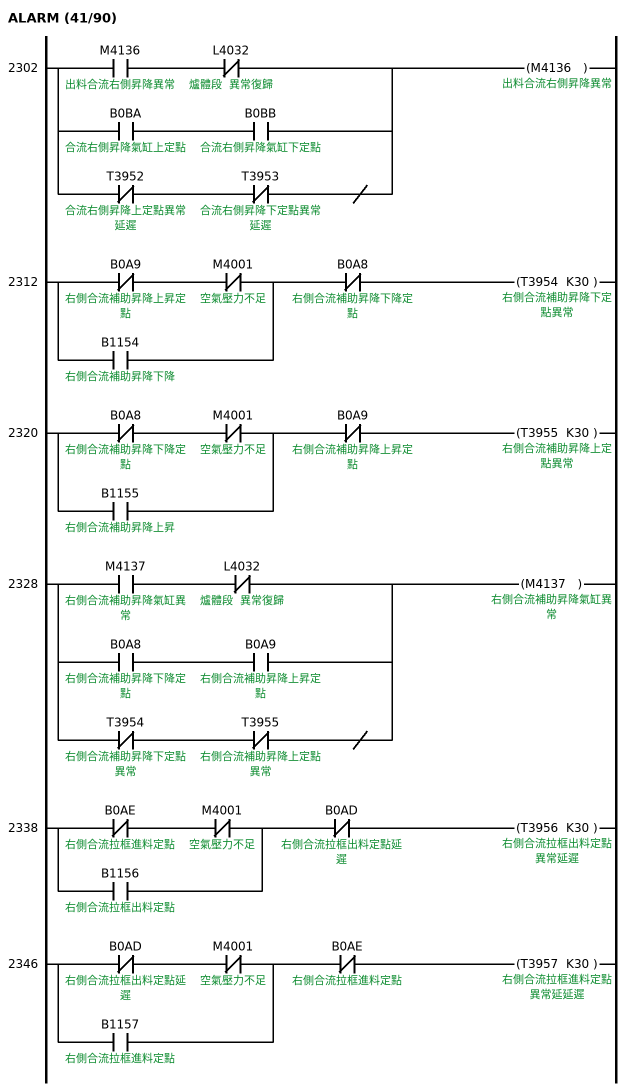
2302  LD      M4136  ; 出料合流右側昇降異常
      ANI     L4032  ; 爐體段  異常復歸
      LD      B0BA  ; 合流右側昇降氣缸上定點
      AND     B0BB  ; 合流右側昇降氣缸下定點
      ORB
      LDI     T3952  ; 合流右側昇降上定點異常延遲
      ANI     T3953  ; 合流右側昇降下定點異常延遲
      INV
      ORB
      OUT     M4136  ; 出料合流右側昇降異常
2312  LDI     B0A9  ; 右側合流補助昇降上昇定點
      ANI     M4001  ; 空氣壓力不足
      OR      B1154  ; 右側合流補助昇降下降
      ANI     B0A8  ; 右側合流補助昇降下降定點
      OUT     T3954 K30  ; 右側合流補助昇降下定點異常
2320  LDI     B0A8  ; 右側合流補助昇降下降定點
      ANI     M4001  ; 空氣壓力不足
      OR      B1155  ; 右側合流補助昇降上昇
      ANI     B0A9  ; 右側合流補助昇降上昇定點
      OUT     T3955 K30  ; 右側合流補助昇降上定點異常
2328  LD      M4137  ; 右側合流補助昇降氣缸異常
      ANI     L4032  ; 爐體段  異常復歸
      LD      B0A8  ; 右側合流補助昇降下降定點
      AND     B0A9  ; 右側合流補助昇降上昇定點
      ORB
      LDI     T3954  ; 右側合流補助昇降下定點異常
      ANI     T3955  ; 右側合流補助昇降上定點異常
      INV
      ORB
      OUT     M4137  ; 右側合流補助昇降氣缸異常
2338  LDI     B0AE  ; 右側合流拉框進料定點
      ANI     M4001  ; 空氣壓力不足
      OR      B1156  ; 右側合流拉框出料定點
      ANI     B0AD  ; 右側合流拉框出料定點延遲
      OUT     T3956 K30  ; 右側合流拉框出料定點異常延遲
2346  LDI     B0AD  ; 右側合流拉框出料定點延遲
      ANI     M4001  ; 空氣壓力不足
      OR      B1157  ; 右側合流拉框進料定點
      ANI     B0AE  ; 右側合流拉框進料定點
      OUT     T3957 K30  ; 右側合流拉框進料定點異常延延遲
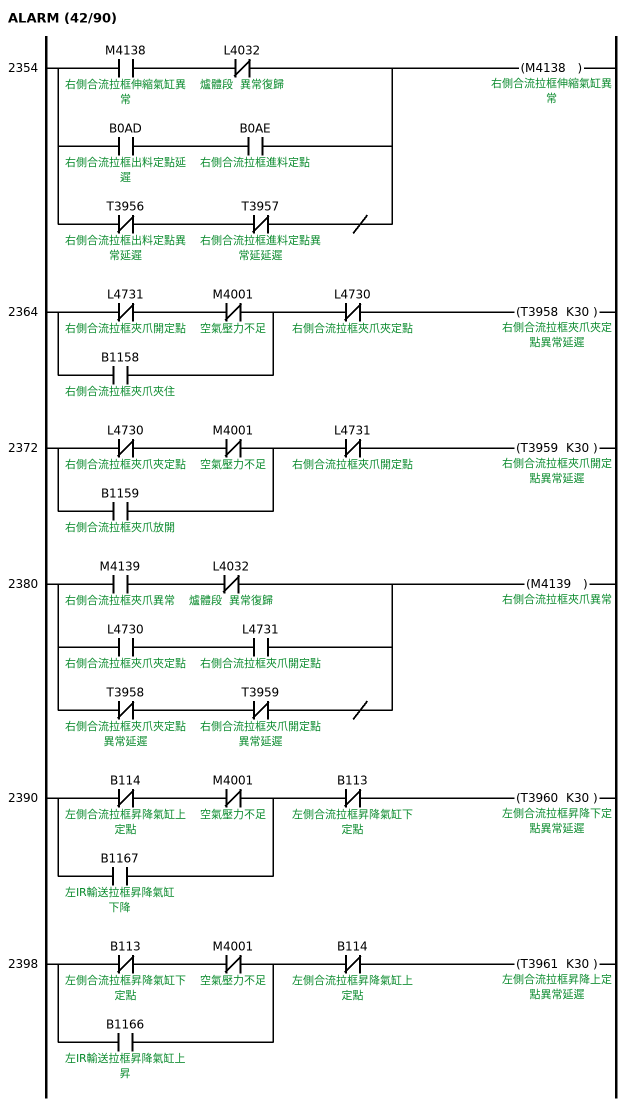
2354  LD      M4138  ; 右側合流拉框伸縮氣缸異常
      ANI     L4032  ; 爐體段  異常復歸
      LD      B0AD  ; 右側合流拉框出料定點延遲
      AND     B0AE  ; 右側合流拉框進料定點
      ORB
      LDI     T3956  ; 右側合流拉框出料定點異常延遲
      ANI     T3957  ; 右側合流拉框進料定點異常延延遲
      INV
      ORB
      OUT     M4138  ; 右側合流拉框伸縮氣缸異常
2364  LDI     L4731  ; 右側合流拉框夾爪開定點
      ANI     M4001  ; 空氣壓力不足
      OR      B1158  ; 右側合流拉框夾爪夾住
      ANI     L4730  ; 右側合流拉框夾爪夾定點
      OUT     T3958 K30  ; 右側合流拉框夾爪夾定點異常延遲
2372  LDI     L4730  ; 右側合流拉框夾爪夾定點
      ANI     M4001  ; 空氣壓力不足
      OR      B1159  ; 右側合流拉框夾爪放開
      ANI     L4731  ; 右側合流拉框夾爪開定點
      OUT     T3959 K30  ; 右側合流拉框夾爪開定點異常延遲
2380  LD      M4139  ; 右側合流拉框夾爪異常
      ANI     L4032  ; 爐體段  異常復歸
      LD      L4730  ; 右側合流拉框夾爪夾定點
      AND     L4731  ; 右側合流拉框夾爪開定點
      ORB
      LDI     T3958  ; 右側合流拉框夾爪夾定點異常延遲
      ANI     T3959  ; 右側合流拉框夾爪開定點異常延遲
      INV
      ORB
      OUT     M4139  ; 右側合流拉框夾爪異常
2390  LDI     B114  ; 左側合流拉框昇降氣缸上定點
      ANI     M4001  ; 空氣壓力不足
      OR      B1167  ; 左IR輸送拉框昇降氣缸  下降
      ANI     B113  ; 左側合流拉框昇降氣缸下定點
      OUT     T3960 K30  ; 左側合流拉框昇降下定點異常延遲
2398  LDI     B113  ; 左側合流拉框昇降氣缸下定點
      ANI     M4001  ; 空氣壓力不足
      OR      B1166  ; 左IR輸送拉框昇降氣缸上昇
      ANI     B114  ; 左側合流拉框昇降氣缸上定點
      OUT     T3961 K30  ; 左側合流拉框昇降上定點異常延遲
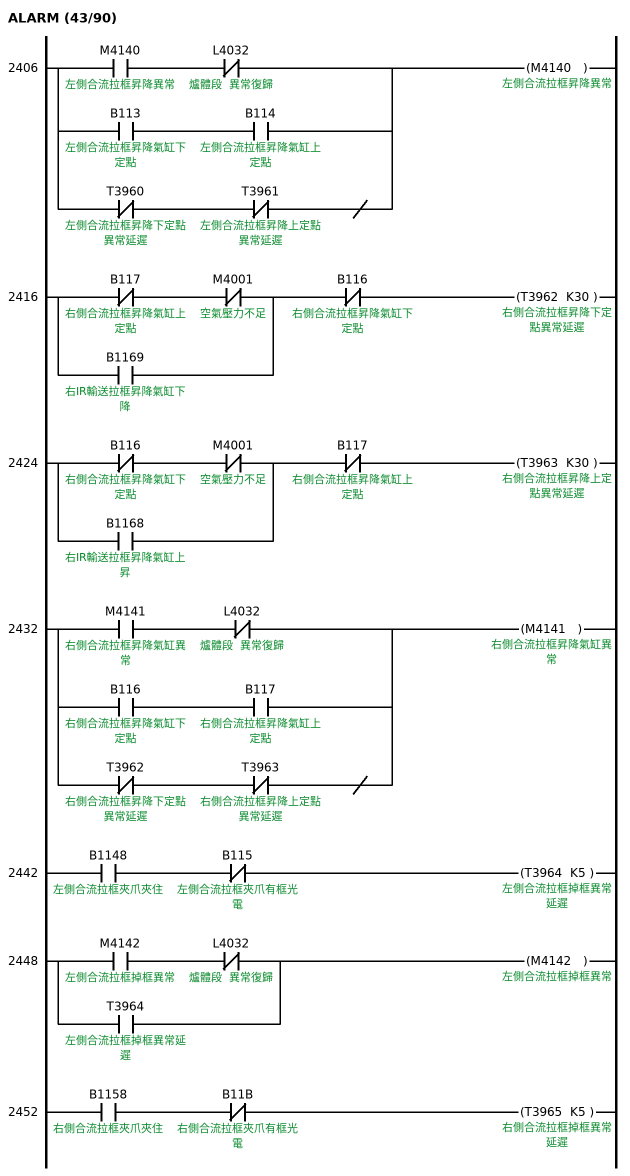
2406  LD      M4140  ; 左側合流拉框昇降異常
      ANI     L4032  ; 爐體段  異常復歸
      LD      B113  ; 左側合流拉框昇降氣缸下定點
      AND     B114  ; 左側合流拉框昇降氣缸上定點
      ORB
      LDI     T3960  ; 左側合流拉框昇降下定點異常延遲
      ANI     T3961  ; 左側合流拉框昇降上定點異常延遲
      INV
      ORB
      OUT     M4140  ; 左側合流拉框昇降異常
2416  LDI     B117  ; 右側合流拉框昇降氣缸上定點
      ANI     M4001  ; 空氣壓力不足
      OR      B1169  ; 右IR輸送拉框昇降氣缸下降
      ANI     B116  ; 右側合流拉框昇降氣缸下定點
      OUT     T3962 K30  ; 右側合流拉框昇降下定點異常延遲
2424  LDI     B116  ; 右側合流拉框昇降氣缸下定點
      ANI     M4001  ; 空氣壓力不足
      OR      B1168  ; 右IR輸送拉框昇降氣缸上昇
      ANI     B117  ; 右側合流拉框昇降氣缸上定點
      OUT     T3963 K30  ; 右側合流拉框昇降上定點異常延遲
2432  LD      M4141  ; 右側合流拉框昇降氣缸異常
      ANI     L4032  ; 爐體段  異常復歸
      LD      B116  ; 右側合流拉框昇降氣缸下定點
      AND     B117  ; 右側合流拉框昇降氣缸上定點
      ORB
      LDI     T3962  ; 右側合流拉框昇降下定點異常延遲
      ANI     T3963  ; 右側合流拉框昇降上定點異常延遲
      INV
      ORB
      OUT     M4141  ; 右側合流拉框昇降氣缸異常
2442  LD      B1148  ; 左側合流拉框夾爪夾住
      ANI     B115  ; 左側合流拉框夾爪有框光電
      OUT     T3964 K5  ; 左側合流拉框掉框異常延遲
2448  LD      M4142  ; 左側合流拉框掉框異常
      ANI     L4032  ; 爐體段  異常復歸
      OR      T3964  ; 左側合流拉框掉框異常延遲
      OUT     M4142  ; 左側合流拉框掉框異常
2452  LD      B1158  ; 右側合流拉框夾爪夾住
      ANI     B11B  ; 右側合流拉框夾爪有框光電
      OUT     T3965 K5  ; 右側合流拉框掉框異常延遲
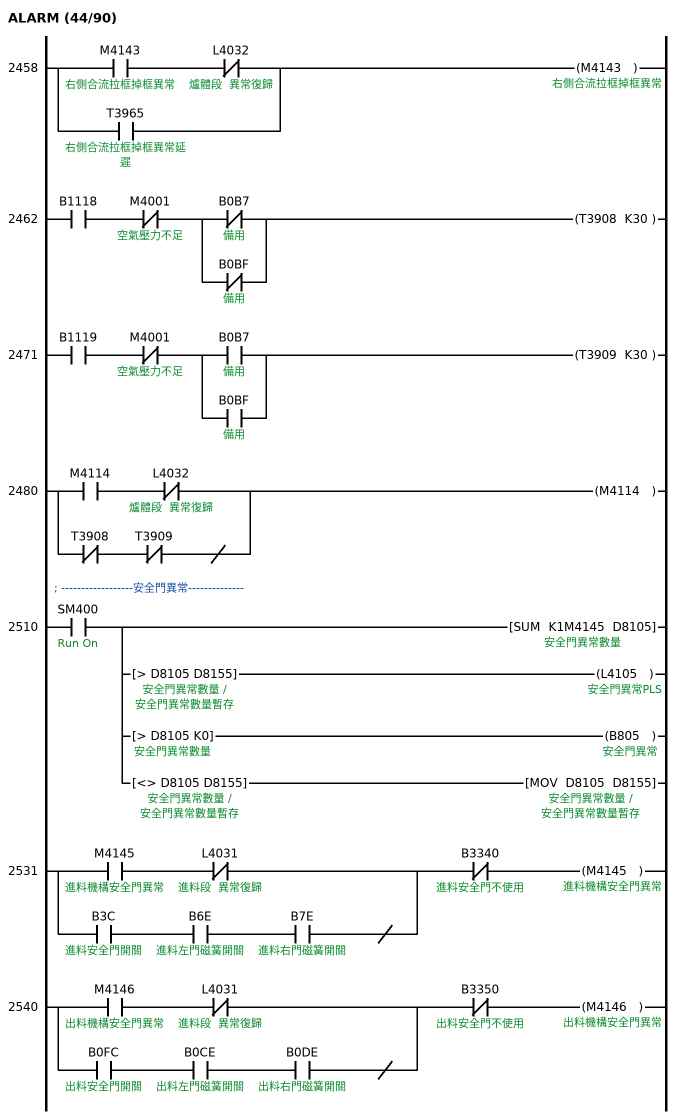
2458  LD      M4143  ; 右側合流拉框掉框異常
      ANI     L4032  ; 爐體段  異常復歸
      OR      T3965  ; 右側合流拉框掉框異常延遲
      OUT     M4143  ; 右側合流拉框掉框異常
2462  LD      B1118
      ANI     M4001  ; 空氣壓力不足
      LDI     B0B7  ; 備用
      ORI     B0BF  ; 備用
      ANB
      OUT     T3908 K30
2471  LD      B1119
      ANI     M4001  ; 空氣壓力不足
      LD      B0B7  ; 備用
      OR      B0BF  ; 備用
      ANB
      OUT     T3909 K30
2480  LD      M4114
      ANI     L4032  ; 爐體段  異常復歸
      LDI     T3908
      ANI     T3909
      INV
      ORB
      OUT     M4114
; ------------------安全門異常--------------
2510  LD      SM400  ; Run On
      SUM     K1M4145 D8105  ; 進料機構安全門異常 / 安全門異常數量
      MPS
      AND>    D8105 D8155  ; 安全門異常數量 / 安全門異常數量暫存
      OUT     L4105  ; 安全門異常PLS
      MRD
      AND>    D8105 K0  ; 安全門異常數量
      OUT     B805  ; 安全門異常
      MPP
      AND<>   D8105 D8155  ; 安全門異常數量 / 安全門異常數量暫存
      MOV     D8105 D8155
2531  LD      M4145  ; 進料機構安全門異常
      ANI     L4031  ; 進料段  異常復歸
      LD      B3C  ; 進料安全門開關
      AND     B6E  ; 進料左門磁簧開關
      AND     B7E  ; 進料右門磁簧開關
      INV
      ORB
      ANI     B3340  ; 進料安全門不使用
      OUT     M4145  ; 進料機構安全門異常
2540  LD      M4146  ; 出料機構安全門異常
      ANI     L4031  ; 進料段  異常復歸
      LD      B0FC  ; 出料安全門開關
      AND     B0CE  ; 出料左門磁簧開關
      AND     B0DE  ; 出料右門磁簧開關
      INV
      ORB
      ANI     B3350  ; 出料安全門不使用
      OUT     M4146  ; 出料機構安全門異常
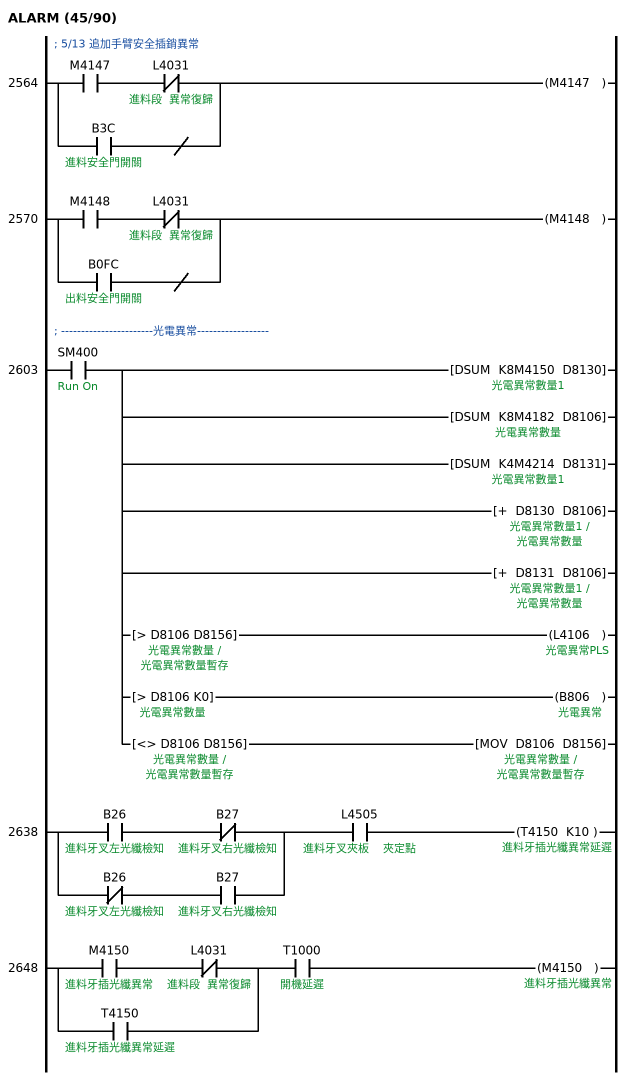
; 5/13 追加手臂安全插銷異常
2564  LD      M4147
      ANI     L4031  ; 進料段  異常復歸
      LD      B3C  ; 進料安全門開關
      INV
      ORB
      OUT     M4147
2570  LD      M4148
      ANI     L4031  ; 進料段  異常復歸
      LD      B0FC  ; 出料安全門開關
      INV
      ORB
      OUT     M4148
; -----------------------光電異常------------------
2603  LD      SM400  ; Run On
      DSUM    K8M4150 D8130  ; 進料牙插光纖異常 / 光電異常數量1
      DSUM    K8M4182 D8106  ; 出料卡板異常 / 光電異常數量
      DSUM    K4M4214 D8131  ; 光電異常數量1
      +       D8130 D8106
      +       D8131 D8106
      MPS
      AND>    D8106 D8156  ; 光電異常數量 / 光電異常數量暫存
      OUT     L4106  ; 光電異常PLS
      MRD
      AND>    D8106 K0  ; 光電異常數量
      OUT     B806  ; 光電異常
      MPP
      AND<>   D8106 D8156  ; 光電異常數量 / 光電異常數量暫存
      MOV     D8106 D8156
2638  LD      B26  ; 進料牙叉左光纖檢知
      ANI     B27  ; 進料牙叉右光纖檢知
      LDI     B26  ; 進料牙叉左光纖檢知
      AND     B27  ; 進料牙叉右光纖檢知
      ORB
      AND     L4505  ; 進料牙叉夾板    夾定點
      OUT     T4150 K10  ; 進料牙插光纖異常延遲
2648  LD      M4150  ; 進料牙插光纖異常
      ANI     L4031  ; 進料段  異常復歸
      OR      T4150  ; 進料牙插光纖異常延遲
      AND     T1000  ; 開機延遲
      OUT     M4150  ; 進料牙插光纖異常
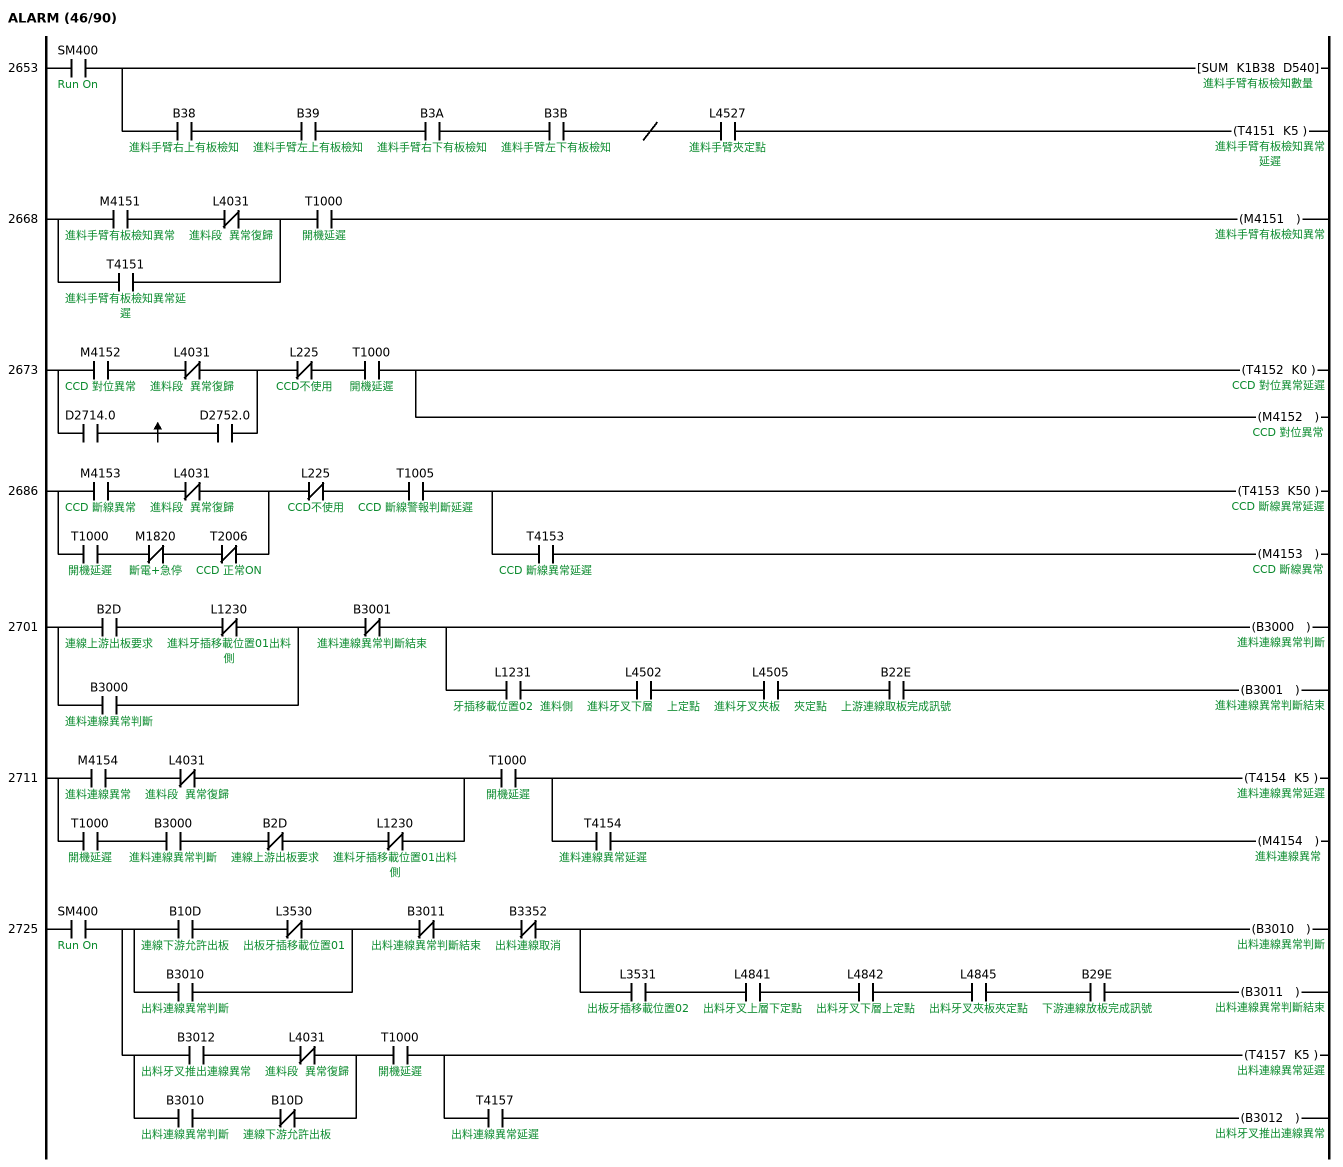
2653  LD      SM400  ; Run On
      SUM     K1B38 D540  ; 進料手臂右上有板檢知 / 進料手臂有板檢知數量
      AND     B38  ; 進料手臂右上有板檢知
      AND     B39  ; 進料手臂左上有板檢知
      AND     B3A  ; 進料手臂右下有板檢知
      AND     B3B  ; 進料手臂左下有板檢知
      INV
      AND     L4527  ; 進料手臂夾定點
      OUT     T4151 K5  ; 進料手臂有板檢知異常延遲
2668  LD      M4151  ; 進料手臂有板檢知異常
      ANI     L4031  ; 進料段  異常復歸
      OR      T4151  ; 進料手臂有板檢知異常延遲
      AND     T1000  ; 開機延遲
      OUT     M4151  ; 進料手臂有板檢知異常
2673  LD      M4152  ; CCD 對位異常
      ANI     L4031  ; 進料段  異常復歸
      LD      D2714.0
      MEP
      AND     D2752.0
      ORB
      ANI     L225  ; CCD不使用
      AND     T1000  ; 開機延遲
      OUT     T4152 K0  ; CCD 對位異常延遲
      OUT     M4152  ; CCD 對位異常
2686  LD      M4153  ; CCD 斷線異常
      ANI     L4031  ; 進料段  異常復歸
      LD      T1000  ; 開機延遲
      ANI     M1820  ; 斷電+急停
      ANI     T2006  ; CCD 正常ON
      ORB
      ANI     L225  ; CCD不使用
      AND     T1005  ; CCD 斷線警報判斷延遲
      OUT     T4153 K50  ; CCD 斷線異常延遲
      AND     T4153  ; CCD 斷線異常延遲
      OUT     M4153  ; CCD 斷線異常
2701  LD      B2D  ; 連線上游出板要求
      ANI     L1230  ; 進料牙插移載位置01出料側
      OR      B3000  ; 進料連線異常判斷
      ANI     B3001  ; 進料連線異常判斷結束
      OUT     B3000  ; 進料連線異常判斷
      AND     L1231  ; 牙插移載位置02  進料側
      AND     L4502  ; 進料牙叉下層    上定點
      AND     L4505  ; 進料牙叉夾板    夾定點
      AND     B22E  ; 上游連線取板完成訊號
      OUT     B3001  ; 進料連線異常判斷結束
2711  LD      M4154  ; 進料連線異常
      ANI     L4031  ; 進料段  異常復歸
      LD      T1000  ; 開機延遲
      AND     B3000  ; 進料連線異常判斷
      ANI     B2D  ; 連線上游出板要求
      ANI     L1230  ; 進料牙插移載位置01出料側
      ORB
      AND     T1000  ; 開機延遲
      OUT     T4154 K5  ; 進料連線異常延遲
      AND     T4154  ; 進料連線異常延遲
      OUT     M4154  ; 進料連線異常
2725  LD      SM400  ; Run On
      MPS
      LD      B10D  ; 連線下游允許出板
      ANI     L3530  ; 出板牙插移載位置01
      OR      B3010  ; 出料連線異常判斷
      ANB
      ANI     B3011  ; 出料連線異常判斷結束
      ANI     B3352  ; 出料連線取消
      OUT     B3010  ; 出料連線異常判斷
      AND     L3531  ; 出板牙插移載位置02
      AND     L4841  ; 出料牙叉上層下定點
      AND     L4842  ; 出料牙叉下層上定點
      AND     L4845  ; 出料牙叉夾板夾定點
      AND     B29E  ; 下游連線放板完成訊號
      OUT     B3011  ; 出料連線異常判斷結束
      MPP
      LD      B3012  ; 出料牙叉推出連線異常
      ANI     L4031  ; 進料段  異常復歸
      LD      B3010  ; 出料連線異常判斷
      ANI     B10D  ; 連線下游允許出板
      ORB
      ANB
      AND     T1000  ; 開機延遲
      OUT     T4157 K5  ; 出料連線異常延遲
      AND     T4157  ; 出料連線異常延遲
      OUT     B3012  ; 出料牙叉推出連線異常
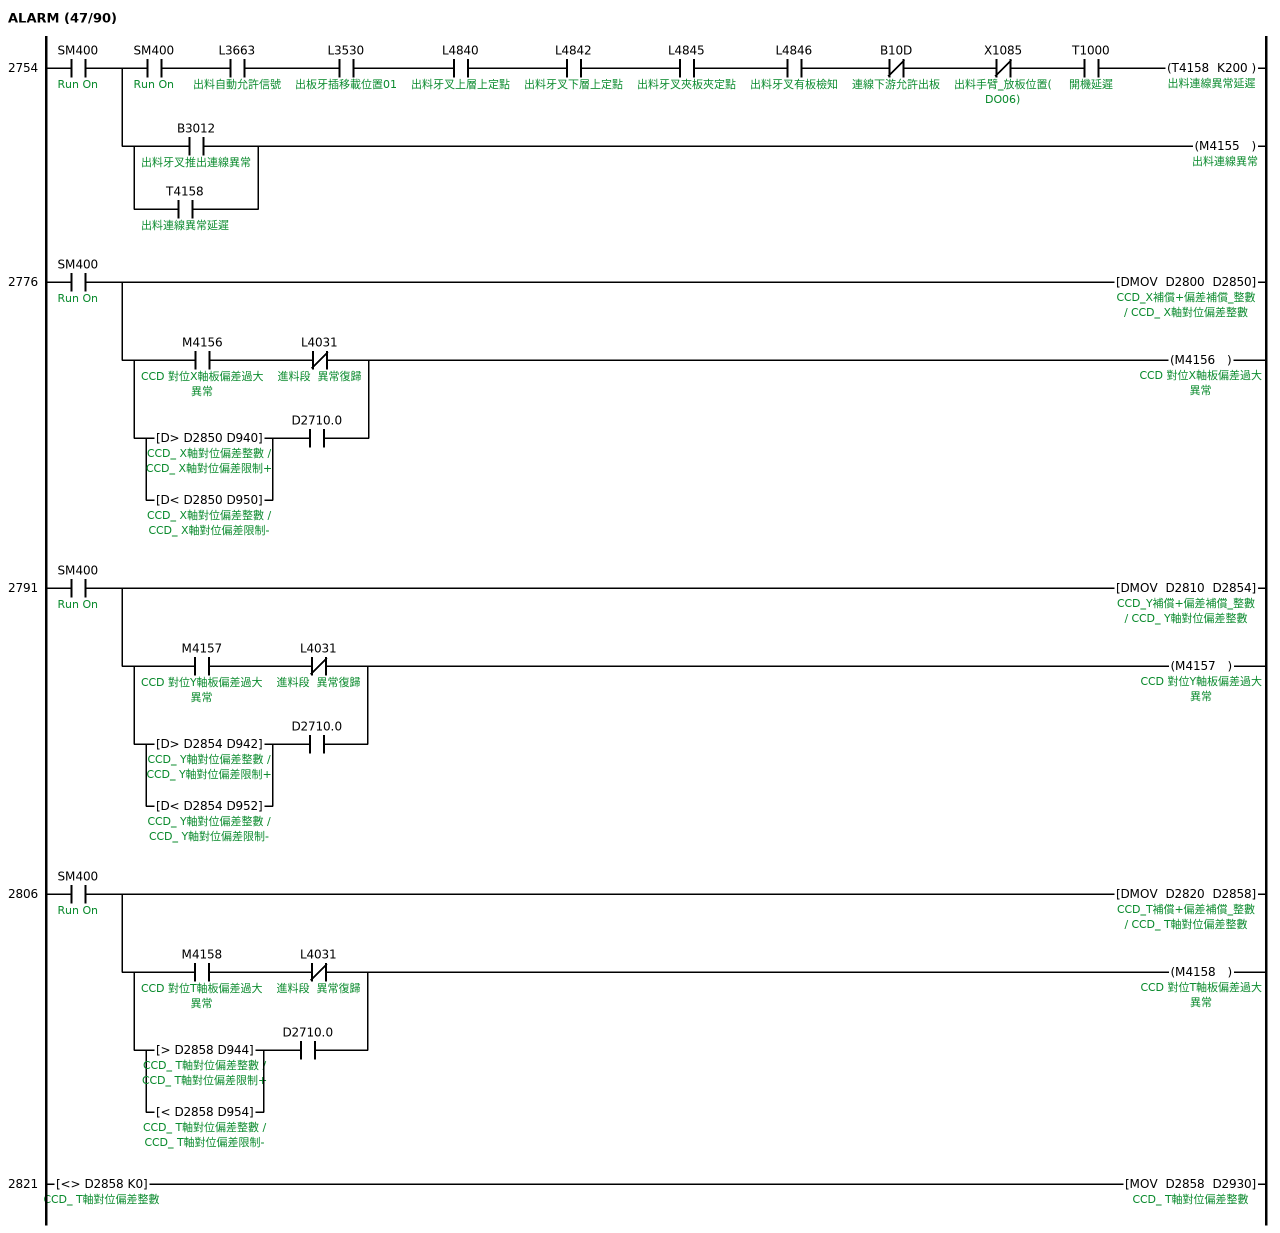
2754  LD      SM400  ; Run On
      MPS
      AND     SM400  ; Run On
      AND     L3663  ; 出料自動允許信號
      AND     L3530  ; 出板牙插移載位置01
      AND     L4840  ; 出料牙叉上層上定點
      AND     L4842  ; 出料牙叉下層上定點
      AND     L4845  ; 出料牙叉夾板夾定點
      AND     L4846  ; 出料牙叉有板檢知
      ANI     B10D  ; 連線下游允許出板
      ANI     X1085  ; 出料手臂_放板位置(DO06)
      AND     T1000  ; 開機延遲
      OUT     T4158 K200  ; 出料連線異常延遲
      MPP
      LD      B3012  ; 出料牙叉推出連線異常
      OR      T4158  ; 出料連線異常延遲
      ANB
      OUT     M4155  ; 出料連線異常
2776  LD      SM400  ; Run On
      DMOV    D2800 D2850  ; CCD_X補償+偏差補償_整數 / CCD_ X軸對位偏差整數
      LD      M4156  ; CCD 對位X軸板偏差過大異常
      ANI     L4031  ; 進料段  異常復歸
      LDD>    D2850 D940  ; CCD_ X軸對位偏差整數 / CCD_ X軸對位偏差限制+
      ORD<    D2850 D950  ; CCD_ X軸對位偏差整數 / CCD_ X軸對位偏差限制-
      AND     D2710.0
      ORB
      ANB
      OUT     M4156  ; CCD 對位X軸板偏差過大異常
2791  LD      SM400  ; Run On
      DMOV    D2810 D2854  ; CCD_Y補償+偏差補償_整數 / CCD_ Y軸對位偏差整數
      LD      M4157  ; CCD 對位Y軸板偏差過大異常
      ANI     L4031  ; 進料段  異常復歸
      LDD>    D2854 D942  ; CCD_ Y軸對位偏差整數 / CCD_ Y軸對位偏差限制+
      ORD<    D2854 D952  ; CCD_ Y軸對位偏差整數 / CCD_ Y軸對位偏差限制-
      AND     D2710.0
      ORB
      ANB
      OUT     M4157  ; CCD 對位Y軸板偏差過大異常
2806  LD      SM400  ; Run On
      DMOV    D2820 D2858  ; CCD_T補償+偏差補償_整數 / CCD_ T軸對位偏差整數
      LD      M4158  ; CCD 對位T軸板偏差過大異常
      ANI     L4031  ; 進料段  異常復歸
      LD>     D2858 D944  ; CCD_ T軸對位偏差整數 / CCD_ T軸對位偏差限制+
      OR<     D2858 D954  ; CCD_ T軸對位偏差整數 / CCD_ T軸對位偏差限制-
      AND     D2710.0
      ORB
      ANB
      OUT     M4158  ; CCD 對位T軸板偏差過大異常
2821  LD<>    D2858 K0  ; CCD_ T軸對位偏差整數
      MOV     D2858 D2930
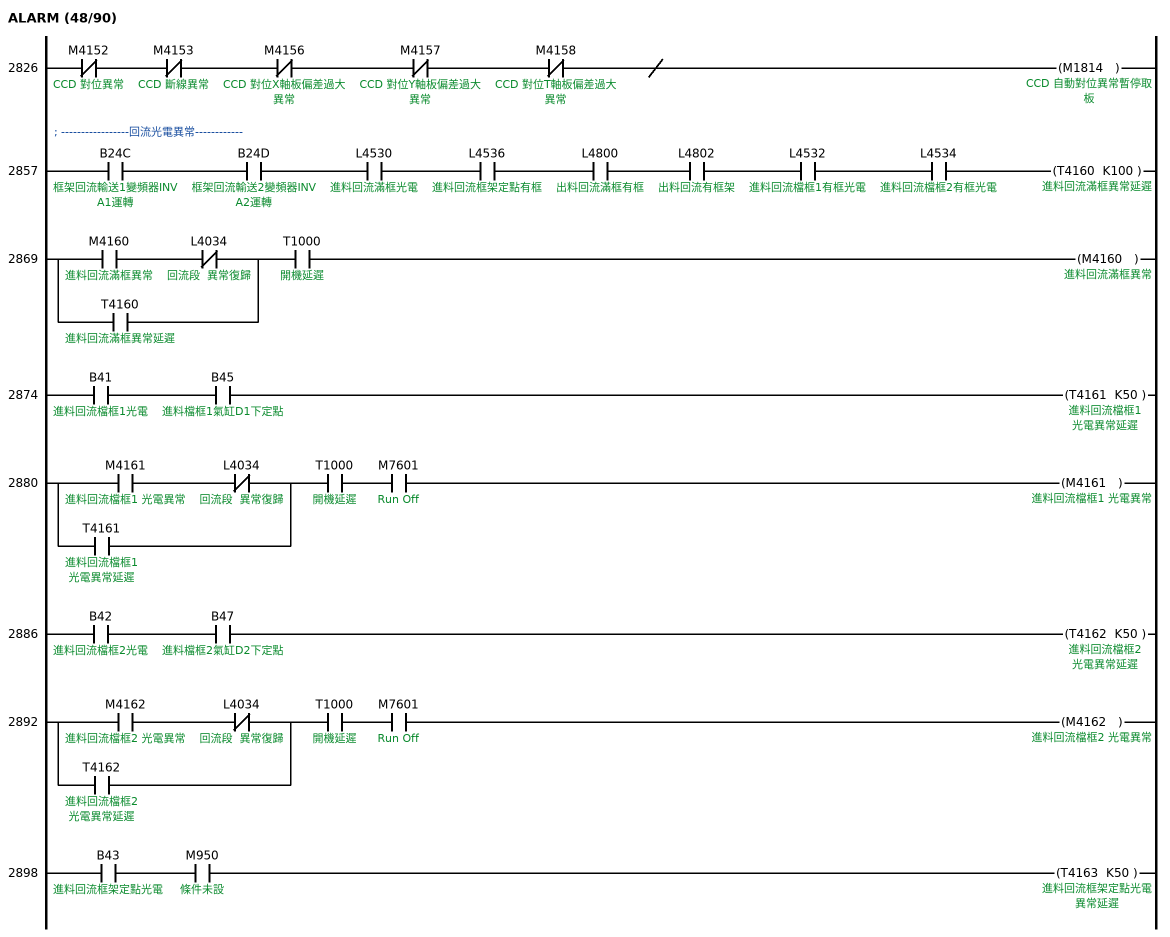
2826  LDI     M4152  ; CCD 對位異常
      ANI     M4153  ; CCD 斷線異常
      ANI     M4156  ; CCD 對位X軸板偏差過大異常
      ANI     M4157  ; CCD 對位Y軸板偏差過大異常
      ANI     M4158  ; CCD 對位T軸板偏差過大異常
      INV
      OUT     M1814  ; CCD 自動對位異常暫停取板
; -----------------回流光電異常------------
2857  LD      B24C  ; 框架回流輸送1變頻器INVA1運轉
      AND     B24D  ; 框架回流輸送2變頻器INVA2運轉
      AND     L4530  ; 進料回流滿框光電
      AND     L4536  ; 進料回流框架定點有框
      AND     L4800  ; 出料回流滿框有框
      AND     L4802  ; 出料回流有框架
      AND     L4532  ; 進料回流檔框1有框光電
      AND     L4534  ; 進料回流檔框2有框光電
      OUT     T4160 K100  ; 進料回流滿框異常延遲
2869  LD      M4160  ; 進料回流滿框異常
      ANI     L4034  ; 回流段  異常復歸
      OR      T4160  ; 進料回流滿框異常延遲
      AND     T1000  ; 開機延遲
      OUT     M4160  ; 進料回流滿框異常
2874  LD      B41  ; 進料回流檔框1光電
      AND     B45  ; 進料檔框1氣缸D1下定點
      OUT     T4161 K50  ; 進料回流檔框1 光電異常延遲
2880  LD      M4161  ; 進料回流檔框1 光電異常
      ANI     L4034  ; 回流段  異常復歸
      OR      T4161  ; 進料回流檔框1 光電異常延遲
      AND     T1000  ; 開機延遲
      AND     M7601  ; Run Off
      OUT     M4161  ; 進料回流檔框1 光電異常
2886  LD      B42  ; 進料回流檔框2光電
      AND     B47  ; 進料檔框2氣缸D2下定點
      OUT     T4162 K50  ; 進料回流檔框2 光電異常延遲
2892  LD      M4162  ; 進料回流檔框2 光電異常
      ANI     L4034  ; 回流段  異常復歸
      OR      T4162  ; 進料回流檔框2 光電異常延遲
      AND     T1000  ; 開機延遲
      AND     M7601  ; Run Off
      OUT     M4162  ; 進料回流檔框2 光電異常
2898  LD      B43  ; 進料回流框架定點光電
      AND     M950  ; 條件未設
      OUT     T4163 K50  ; 進料回流框架定點光電異常延遲
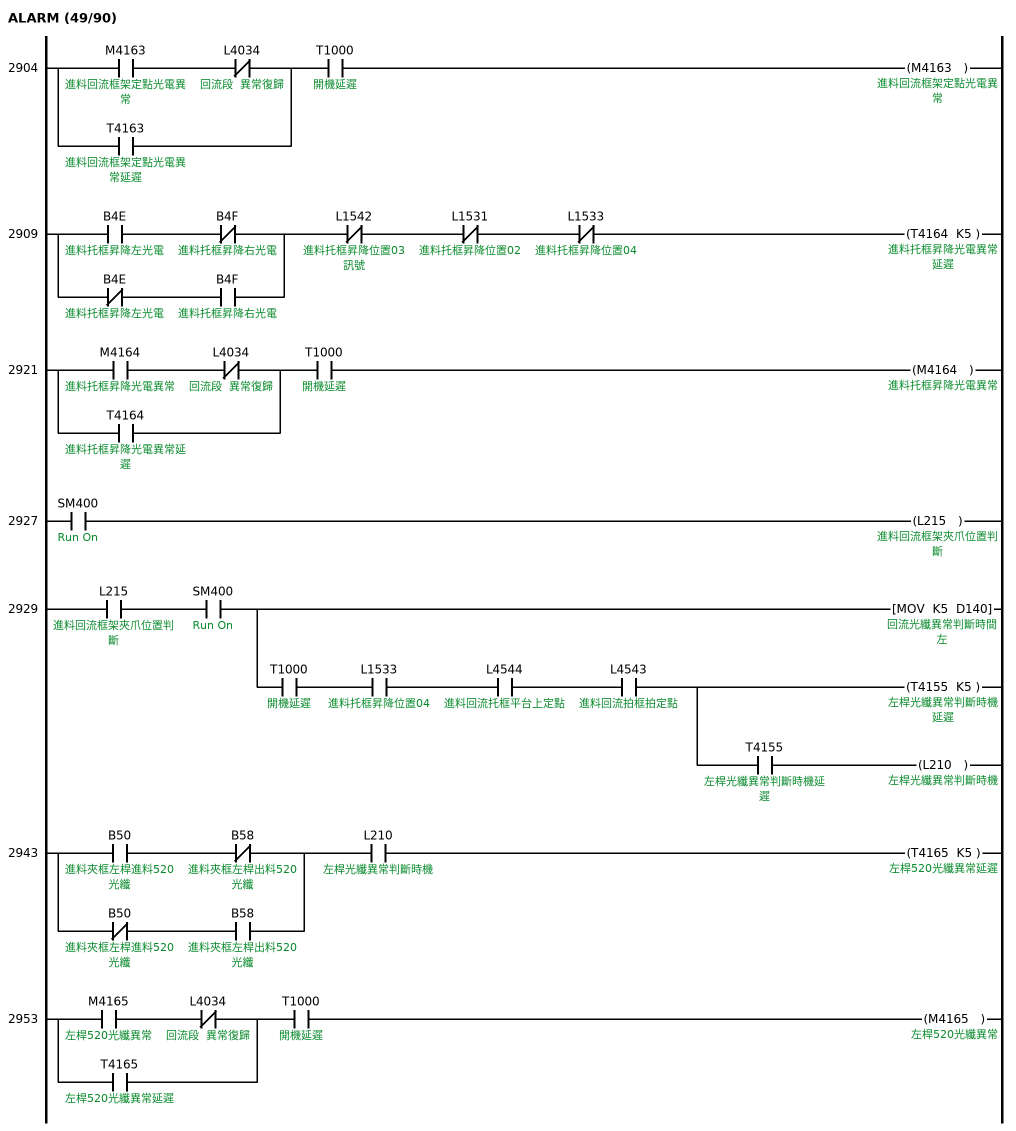
2904  LD      M4163  ; 進料回流框架定點光電異常
      ANI     L4034  ; 回流段  異常復歸
      OR      T4163  ; 進料回流框架定點光電異常延遲
      AND     T1000  ; 開機延遲
      OUT     M4163  ; 進料回流框架定點光電異常
2909  LD      B4E  ; 進料托框昇降左光電
      ANI     B4F  ; 進料托框昇降右光電
      LDI     B4E  ; 進料托框昇降左光電
      AND     B4F  ; 進料托框昇降右光電
      ORB
      ANI     L1542  ; 進料托框昇降位置03 訊號
      ANI     L1531  ; 進料托框昇降位置02
      ANI     L1533  ; 進料托框昇降位置04
      OUT     T4164 K5  ; 進料托框昇降光電異常延遲
2921  LD      M4164  ; 進料托框昇降光電異常
      ANI     L4034  ; 回流段  異常復歸
      OR      T4164  ; 進料托框昇降光電異常延遲
      AND     T1000  ; 開機延遲
      OUT     M4164  ; 進料托框昇降光電異常
2927  LD      SM400  ; Run On
      OUT     L215  ; 進料回流框架夾爪位置判斷
2929  LD      L215  ; 進料回流框架夾爪位置判斷
      AND     SM400  ; Run On
      MOV     K5 D140  ; 回流光纖異常判斷時間左
      AND     T1000  ; 開機延遲
      AND     L1533  ; 進料托框昇降位置04
      AND     L4544  ; 進料回流托框平台上定點
      AND     L4543  ; 進料回流拍框拍定點
      OUT     T4155 K5  ; 左桿光纖異常判斷時機延遲
      AND     T4155  ; 左桿光纖異常判斷時機延遲
      OUT     L210  ; 左桿光纖異常判斷時機
2943  LD      B50  ; 進料夾框左桿進料520 光纖
      ANI     B58  ; 進料夾框左桿出料520 光纖
      LDI     B50  ; 進料夾框左桿進料520 光纖
      AND     B58  ; 進料夾框左桿出料520 光纖
      ORB
      AND     L210  ; 左桿光纖異常判斷時機
      OUT     T4165 K5  ; 左桿520光纖異常延遲
2953  LD      M4165  ; 左桿520光纖異常
      ANI     L4034  ; 回流段  異常復歸
      OR      T4165  ; 左桿520光纖異常延遲
      AND     T1000  ; 開機延遲
      OUT     M4165  ; 左桿520光纖異常
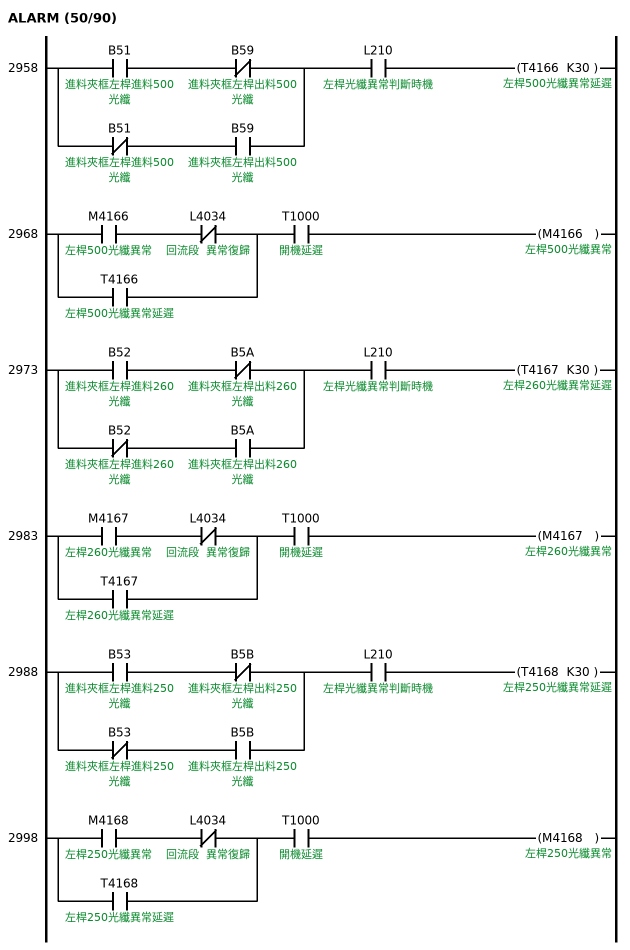
2958  LD      B51  ; 進料夾框左桿進料500 光纖
      ANI     B59  ; 進料夾框左桿出料500 光纖
      LDI     B51  ; 進料夾框左桿進料500 光纖
      AND     B59  ; 進料夾框左桿出料500 光纖
      ORB
      AND     L210  ; 左桿光纖異常判斷時機
      OUT     T4166 K30  ; 左桿500光纖異常延遲
2968  LD      M4166  ; 左桿500光纖異常
      ANI     L4034  ; 回流段  異常復歸
      OR      T4166  ; 左桿500光纖異常延遲
      AND     T1000  ; 開機延遲
      OUT     M4166  ; 左桿500光纖異常
2973  LD      B52  ; 進料夾框左桿進料260 光纖
      ANI     B5A  ; 進料夾框左桿出料260 光纖
      LDI     B52  ; 進料夾框左桿進料260 光纖
      AND     B5A  ; 進料夾框左桿出料260 光纖
      ORB
      AND     L210  ; 左桿光纖異常判斷時機
      OUT     T4167 K30  ; 左桿260光纖異常延遲
2983  LD      M4167  ; 左桿260光纖異常
      ANI     L4034  ; 回流段  異常復歸
      OR      T4167  ; 左桿260光纖異常延遲
      AND     T1000  ; 開機延遲
      OUT     M4167  ; 左桿260光纖異常
2988  LD      B53  ; 進料夾框左桿進料250 光纖
      ANI     B5B  ; 進料夾框左桿出料250 光纖
      LDI     B53  ; 進料夾框左桿進料250 光纖
      AND     B5B  ; 進料夾框左桿出料250 光纖
      ORB
      AND     L210  ; 左桿光纖異常判斷時機
      OUT     T4168 K30  ; 左桿250光纖異常延遲
2998  LD      M4168  ; 左桿250光纖異常
      ANI     L4034  ; 回流段  異常復歸
      OR      T4168  ; 左桿250光纖異常延遲
      AND     T1000  ; 開機延遲
      OUT     M4168  ; 左桿250光纖異常
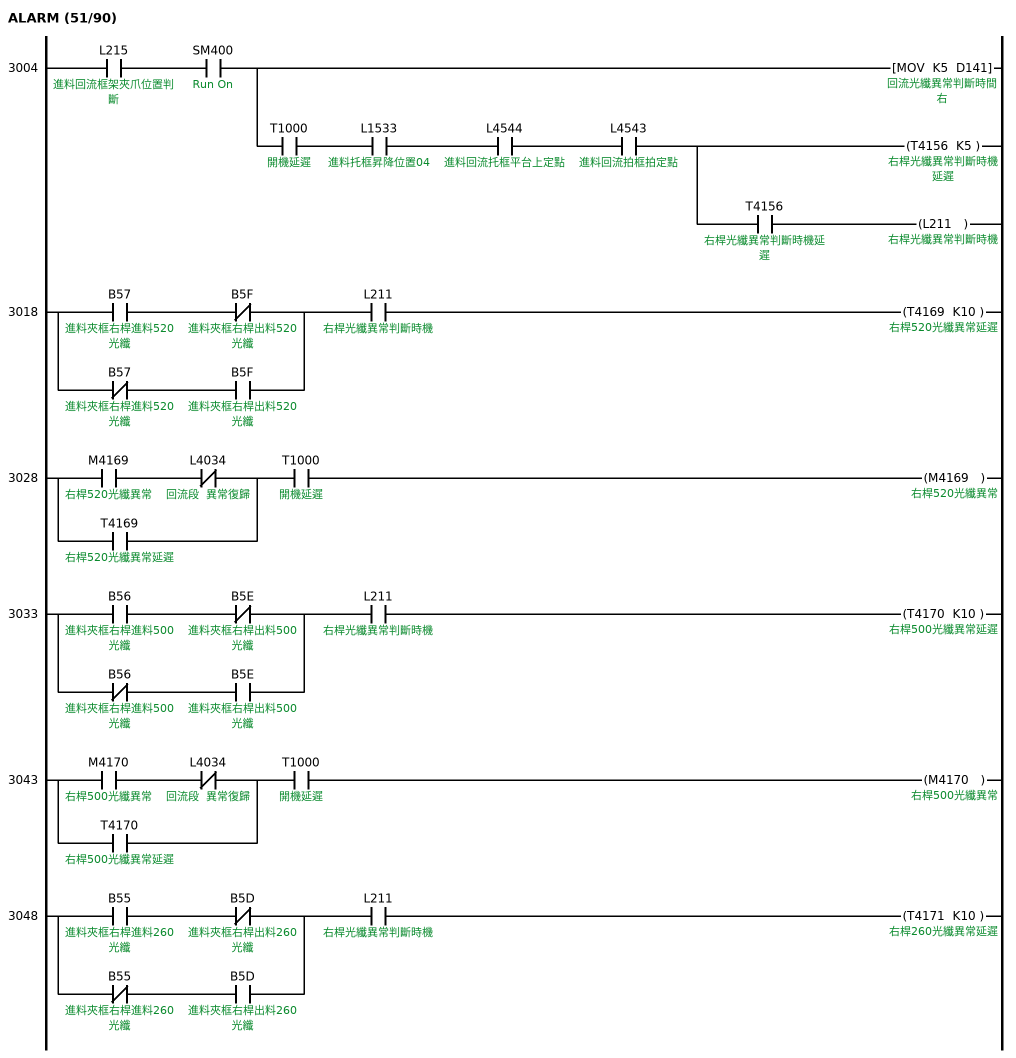
3004  LD      L215  ; 進料回流框架夾爪位置判斷
      AND     SM400  ; Run On
      MOV     K5 D141  ; 回流光纖異常判斷時間右
      AND     T1000  ; 開機延遲
      AND     L1533  ; 進料托框昇降位置04
      AND     L4544  ; 進料回流托框平台上定點
      AND     L4543  ; 進料回流拍框拍定點
      OUT     T4156 K5  ; 右桿光纖異常判斷時機延遲
      AND     T4156  ; 右桿光纖異常判斷時機延遲
      OUT     L211  ; 右桿光纖異常判斷時機
3018  LD      B57  ; 進料夾框右桿進料520 光纖
      ANI     B5F  ; 進料夾框右桿出料520 光纖
      LDI     B57  ; 進料夾框右桿進料520 光纖
      AND     B5F  ; 進料夾框右桿出料520 光纖
      ORB
      AND     L211  ; 右桿光纖異常判斷時機
      OUT     T4169 K10  ; 右桿520光纖異常延遲
3028  LD      M4169  ; 右桿520光纖異常
      ANI     L4034  ; 回流段  異常復歸
      OR      T4169  ; 右桿520光纖異常延遲
      AND     T1000  ; 開機延遲
      OUT     M4169  ; 右桿520光纖異常
3033  LD      B56  ; 進料夾框右桿進料500 光纖
      ANI     B5E  ; 進料夾框右桿出料500 光纖
      LDI     B56  ; 進料夾框右桿進料500 光纖
      AND     B5E  ; 進料夾框右桿出料500 光纖
      ORB
      AND     L211  ; 右桿光纖異常判斷時機
      OUT     T4170 K10  ; 右桿500光纖異常延遲
3043  LD      M4170  ; 右桿500光纖異常
      ANI     L4034  ; 回流段  異常復歸
      OR      T4170  ; 右桿500光纖異常延遲
      AND     T1000  ; 開機延遲
      OUT     M4170  ; 右桿500光纖異常
3048  LD      B55  ; 進料夾框右桿進料260 光纖
      ANI     B5D  ; 進料夾框右桿出料260 光纖
      LDI     B55  ; 進料夾框右桿進料260 光纖
      AND     B5D  ; 進料夾框右桿出料260 光纖
      ORB
      AND     L211  ; 右桿光纖異常判斷時機
      OUT     T4171 K10  ; 右桿260光纖異常延遲
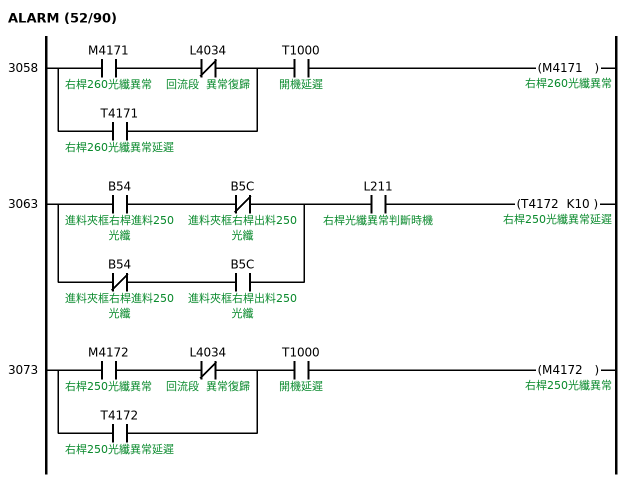
3058  LD      M4171  ; 右桿260光纖異常
      ANI     L4034  ; 回流段  異常復歸
      OR      T4171  ; 右桿260光纖異常延遲
      AND     T1000  ; 開機延遲
      OUT     M4171  ; 右桿260光纖異常
3063  LD      B54  ; 進料夾框右桿進料250 光纖
      ANI     B5C  ; 進料夾框右桿出料250 光纖
      LDI     B54  ; 進料夾框右桿進料250 光纖
      AND     B5C  ; 進料夾框右桿出料250 光纖
      ORB
      AND     L211  ; 右桿光纖異常判斷時機
      OUT     T4172 K10  ; 右桿250光纖異常延遲
3073  LD      M4172  ; 右桿250光纖異常
      ANI     L4034  ; 回流段  異常復歸
      OR      T4172  ; 右桿250光纖異常延遲
      AND     T1000  ; 開機延遲
      OUT     M4172  ; 右桿250光纖異常
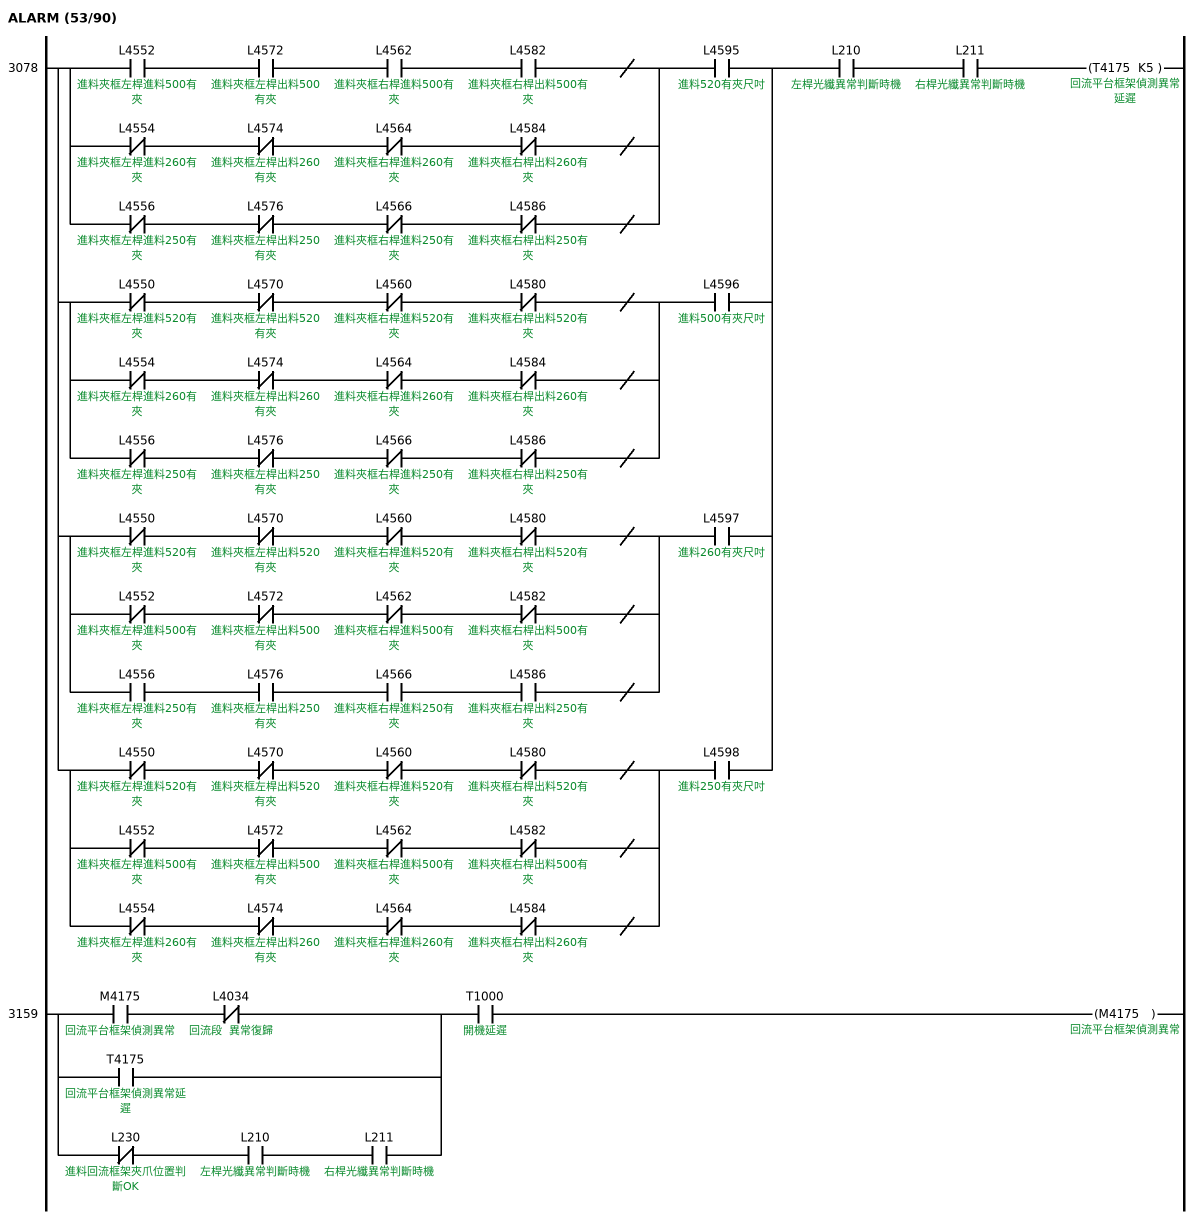
3078  LD      L4552  ; 進料夾框左桿進料500有夾
      AND     L4572  ; 進料夾框左桿出料500 有夾
      AND     L4562  ; 進料夾框右桿進料500有夾
      AND     L4582  ; 進料夾框右桿出料500有夾
      INV
      LDI     L4554  ; 進料夾框左桿進料260有夾
      ANI     L4574  ; 進料夾框左桿出料260 有夾
      ANI     L4564  ; 進料夾框右桿進料260有夾
      ANI     L4584  ; 進料夾框右桿出料260有夾
      INV
      ORB
      LDI     L4556  ; 進料夾框左桿進料250有夾
      ANI     L4576  ; 進料夾框左桿出料250 有夾
      ANI     L4566  ; 進料夾框右桿進料250有夾
      ANI     L4586  ; 進料夾框右桿出料250有夾
      INV
      ORB
      AND     L4595  ; 進料520有夾尺吋
      LDI     L4550  ; 進料夾框左桿進料520有夾
      ANI     L4570  ; 進料夾框左桿出料520 有夾
      ANI     L4560  ; 進料夾框右桿進料520有夾
      ANI     L4580  ; 進料夾框右桿出料520有夾
      INV
      LDI     L4554  ; 進料夾框左桿進料260有夾
      ANI     L4574  ; 進料夾框左桿出料260 有夾
      ANI     L4564  ; 進料夾框右桿進料260有夾
      ANI     L4584  ; 進料夾框右桿出料260有夾
      INV
      ORB
      LDI     L4556  ; 進料夾框左桿進料250有夾
      ANI     L4576  ; 進料夾框左桿出料250 有夾
      ANI     L4566  ; 進料夾框右桿進料250有夾
      ANI     L4586  ; 進料夾框右桿出料250有夾
      INV
      ORB
      AND     L4596  ; 進料500有夾尺吋
      ORB
      LDI     L4550  ; 進料夾框左桿進料520有夾
      ANI     L4570  ; 進料夾框左桿出料520 有夾
      ANI     L4560  ; 進料夾框右桿進料520有夾
      ANI     L4580  ; 進料夾框右桿出料520有夾
      INV
      LDI     L4552  ; 進料夾框左桿進料500有夾
      ANI     L4572  ; 進料夾框左桿出料500 有夾
      ANI     L4562  ; 進料夾框右桿進料500有夾
      ANI     L4582  ; 進料夾框右桿出料500有夾
      INV
      ORB
      LD      L4556  ; 進料夾框左桿進料250有夾
      AND     L4576  ; 進料夾框左桿出料250 有夾
      AND     L4566  ; 進料夾框右桿進料250有夾
      AND     L4586  ; 進料夾框右桿出料250有夾
      INV
      ORB
      AND     L4597  ; 進料260有夾尺吋
      ORB
      LDI     L4550  ; 進料夾框左桿進料520有夾
      ANI     L4570  ; 進料夾框左桿出料520 有夾
      ANI     L4560  ; 進料夾框右桿進料520有夾
      ANI     L4580  ; 進料夾框右桿出料520有夾
      INV
      LDI     L4552  ; 進料夾框左桿進料500有夾
      ANI     L4572  ; 進料夾框左桿出料500 有夾
      ANI     L4562  ; 進料夾框右桿進料500有夾
      ANI     L4582  ; 進料夾框右桿出料500有夾
      INV
      ORB
      LDI     L4554  ; 進料夾框左桿進料260有夾
      ANI     L4574  ; 進料夾框左桿出料260 有夾
      ANI     L4564  ; 進料夾框右桿進料260有夾
      ANI     L4584  ; 進料夾框右桿出料260有夾
      INV
      ORB
      AND     L4598  ; 進料250有夾尺吋
      ORB
      AND     L210  ; 左桿光纖異常判斷時機
      AND     L211  ; 右桿光纖異常判斷時機
      OUT     T4175 K5  ; 回流平台框架偵測異常延遲
3159  LD      M4175  ; 回流平台框架偵測異常
      ANI     L4034  ; 回流段  異常復歸
      OR      T4175  ; 回流平台框架偵測異常延遲
      LDI     L230  ; 進料回流框架夾爪位置判斷OK
      AND     L210  ; 左桿光纖異常判斷時機
      AND     L211  ; 右桿光纖異常判斷時機
      ORB
      AND     T1000  ; 開機延遲
      OUT     M4175  ; 回流平台框架偵測異常
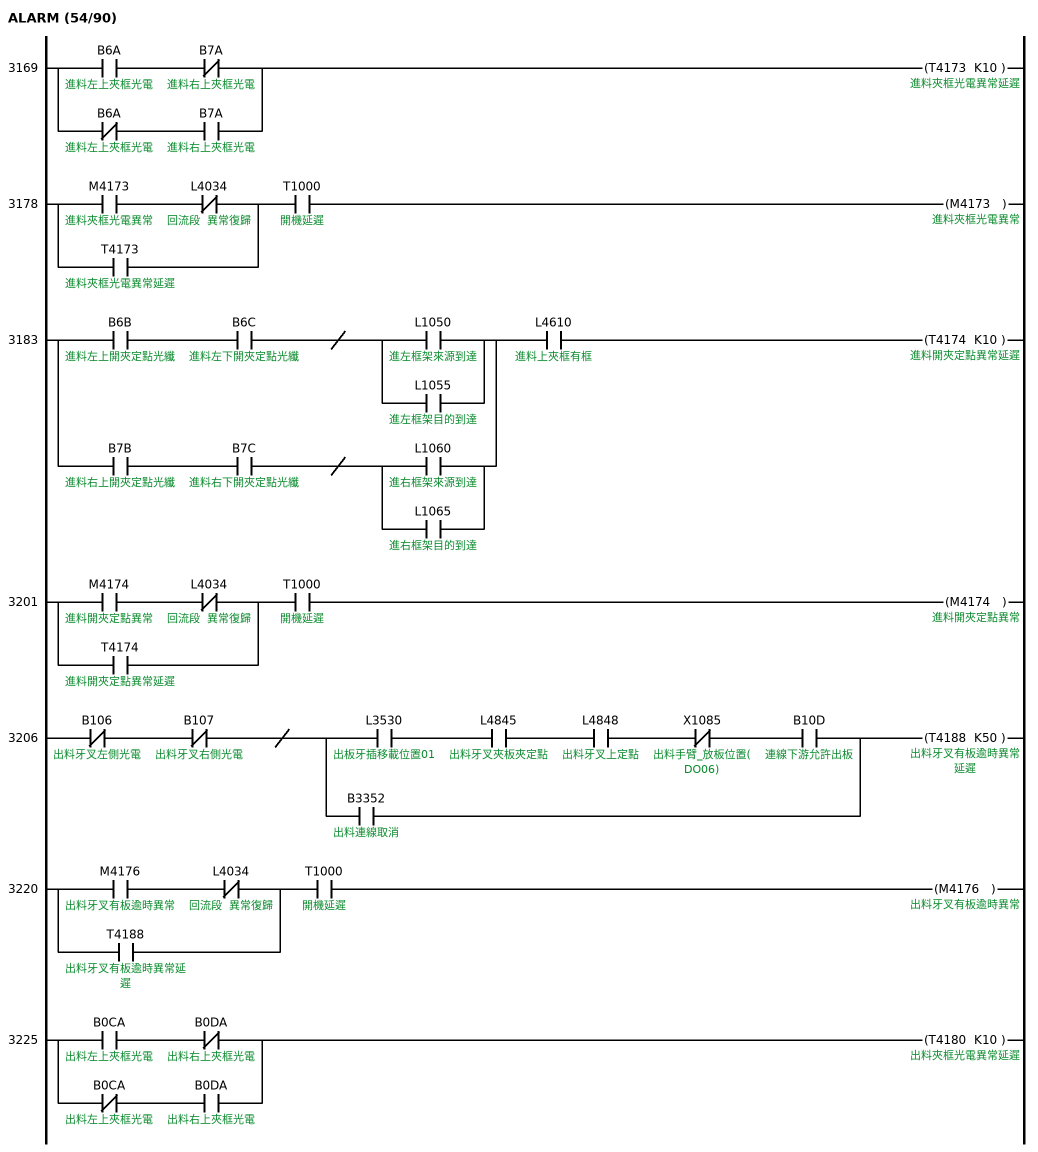
3169  LD      B6A  ; 進料左上夾框光電
      ANI     B7A  ; 進料右上夾框光電
      LDI     B6A  ; 進料左上夾框光電
      AND     B7A  ; 進料右上夾框光電
      ORB
      OUT     T4173 K10  ; 進料夾框光電異常延遲
3178  LD      M4173  ; 進料夾框光電異常
      ANI     L4034  ; 回流段  異常復歸
      OR      T4173  ; 進料夾框光電異常延遲
      AND     T1000  ; 開機延遲
      OUT     M4173  ; 進料夾框光電異常
3183  LD      B6B  ; 進料左上開夾定點光纖
      AND     B6C  ; 進料左下開夾定點光纖
      INV
      LD      L1050  ; 進左框架來源到達
      OR      L1055  ; 進左框架目的到達
      ANB
      LD      B7B  ; 進料右上開夾定點光纖
      AND     B7C  ; 進料右下開夾定點光纖
      INV
      LD      L1060  ; 進右框架來源到達
      OR      L1065  ; 進右框架目的到達
      ANB
      ORB
      AND     L4610  ; 進料上夾框有框
      OUT     T4174 K10  ; 進料開夾定點異常延遲
3201  LD      M4174  ; 進料開夾定點異常
      ANI     L4034  ; 回流段  異常復歸
      OR      T4174  ; 進料開夾定點異常延遲
      AND     T1000  ; 開機延遲
      OUT     M4174  ; 進料開夾定點異常
3206  LDI     B106  ; 出料牙叉左側光電
      ANI     B107  ; 出料牙叉右側光電
      INV
      LD      L3530  ; 出板牙插移載位置01
      AND     L4845  ; 出料牙叉夾板夾定點
      AND     L4848  ; 出料牙叉上定點
      ANI     X1085  ; 出料手臂_放板位置(DO06)
      AND     B10D  ; 連線下游允許出板
      OR      B3352  ; 出料連線取消
      ANB
      OUT     T4188 K50  ; 出料牙叉有板逾時異常延遲
3220  LD      M4176  ; 出料牙叉有板逾時異常
      ANI     L4034  ; 回流段  異常復歸
      OR      T4188  ; 出料牙叉有板逾時異常延遲
      AND     T1000  ; 開機延遲
      OUT     M4176  ; 出料牙叉有板逾時異常
3225  LD      B0CA  ; 出料左上夾框光電
      ANI     B0DA  ; 出料右上夾框光電
      LDI     B0CA  ; 出料左上夾框光電
      AND     B0DA  ; 出料右上夾框光電
      ORB
      OUT     T4180 K10  ; 出料夾框光電異常延遲
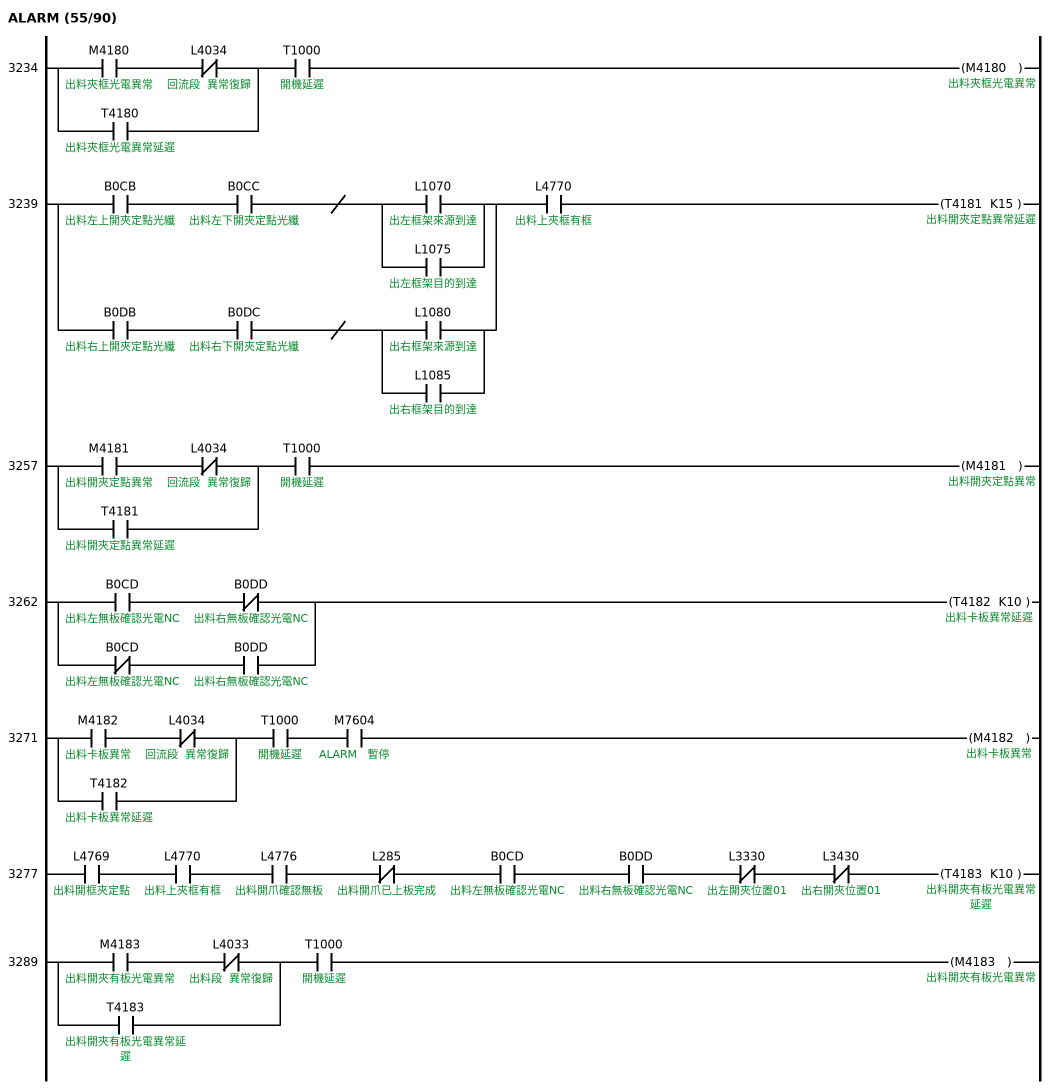
3234  LD      M4180  ; 出料夾框光電異常
      ANI     L4034  ; 回流段  異常復歸
      OR      T4180  ; 出料夾框光電異常延遲
      AND     T1000  ; 開機延遲
      OUT     M4180  ; 出料夾框光電異常
3239  LD      B0CB  ; 出料左上開夾定點光纖
      AND     B0CC  ; 出料左下開夾定點光纖
      INV
      LD      L1070  ; 出左框架來源到達
      OR      L1075  ; 出左框架目的到達
      ANB
      LD      B0DB  ; 出料右上開夾定點光纖
      AND     B0DC  ; 出料右下開夾定點光纖
      INV
      LD      L1080  ; 出右框架來源到達
      OR      L1085  ; 出右框架目的到達
      ANB
      ORB
      AND     L4770  ; 出料上夾框有框
      OUT     T4181 K15  ; 出料開夾定點異常延遲
3257  LD      M4181  ; 出料開夾定點異常
      ANI     L4034  ; 回流段  異常復歸
      OR      T4181  ; 出料開夾定點異常延遲
      AND     T1000  ; 開機延遲
      OUT     M4181  ; 出料開夾定點異常
3262  LD      B0CD  ; 出料左無板確認光電NC
      ANI     B0DD  ; 出料右無板確認光電NC
      LDI     B0CD  ; 出料左無板確認光電NC
      AND     B0DD  ; 出料右無板確認光電NC
      ORB
      OUT     T4182 K10  ; 出料卡板異常延遲
3271  LD      M4182  ; 出料卡板異常
      ANI     L4034  ; 回流段  異常復歸
      OR      T4182  ; 出料卡板異常延遲
      AND     T1000  ; 開機延遲
      AND     M7604  ; ALARM   暫停
      OUT     M4182  ; 出料卡板異常
3277  LD      L4769  ; 出料開框夾定點
      AND     L4770  ; 出料上夾框有框
      AND     L4776  ; 出料開爪確認無板
      ANI     L285  ; 出料開爪已上板完成
      AND     B0CD  ; 出料左無板確認光電NC
      AND     B0DD  ; 出料右無板確認光電NC
      ANI     L3330  ; 出左開夾位置01
      ANI     L3430  ; 出右開夾位置01
      OUT     T4183 K10  ; 出料開夾有板光電異常延遲
3289  LD      M4183  ; 出料開夾有板光電異常
      ANI     L4033  ; 出料段  異常復歸
      OR      T4183  ; 出料開夾有板光電異常延遲
      AND     T1000  ; 開機延遲
      OUT     M4183  ; 出料開夾有板光電異常
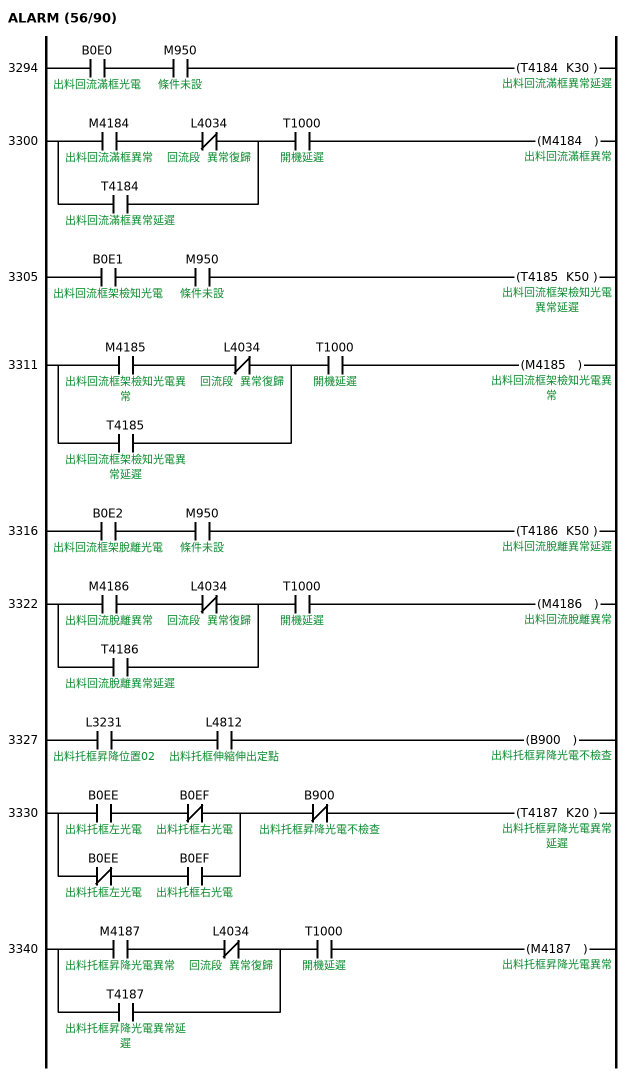
3294  LD      B0E0  ; 出料回流滿框光電
      AND     M950  ; 條件未設
      OUT     T4184 K30  ; 出料回流滿框異常延遲
3300  LD      M4184  ; 出料回流滿框異常
      ANI     L4034  ; 回流段  異常復歸
      OR      T4184  ; 出料回流滿框異常延遲
      AND     T1000  ; 開機延遲
      OUT     M4184  ; 出料回流滿框異常
3305  LD      B0E1  ; 出料回流框架檢知光電
      AND     M950  ; 條件未設
      OUT     T4185 K50  ; 出料回流框架檢知光電異常延遲
3311  LD      M4185  ; 出料回流框架檢知光電異常
      ANI     L4034  ; 回流段  異常復歸
      OR      T4185  ; 出料回流框架檢知光電異常延遲
      AND     T1000  ; 開機延遲
      OUT     M4185  ; 出料回流框架檢知光電異常
3316  LD      B0E2  ; 出料回流框架脫離光電
      AND     M950  ; 條件未設
      OUT     T4186 K50  ; 出料回流脫離異常延遲
3322  LD      M4186  ; 出料回流脫離異常
      ANI     L4034  ; 回流段  異常復歸
      OR      T4186  ; 出料回流脫離異常延遲
      AND     T1000  ; 開機延遲
      OUT     M4186  ; 出料回流脫離異常
3327  LD      L3231  ; 出料托框昇降位置02
      AND     L4812  ; 出料托框伸縮伸出定點
      OUT     B900  ; 出料托框昇降光電不檢查
3330  LD      B0EE  ; 出料托框左光電
      ANI     B0EF  ; 出料托框右光電
      LDI     B0EE  ; 出料托框左光電
      AND     B0EF  ; 出料托框右光電
      ORB
      ANI     B900  ; 出料托框昇降光電不檢查
      OUT     T4187 K20  ; 出料托框昇降光電異常延遲
3340  LD      M4187  ; 出料托框昇降光電異常
      ANI     L4034  ; 回流段  異常復歸
      OR      T4187  ; 出料托框昇降光電異常延遲
      AND     T1000  ; 開機延遲
      OUT     M4187  ; 出料托框昇降光電異常
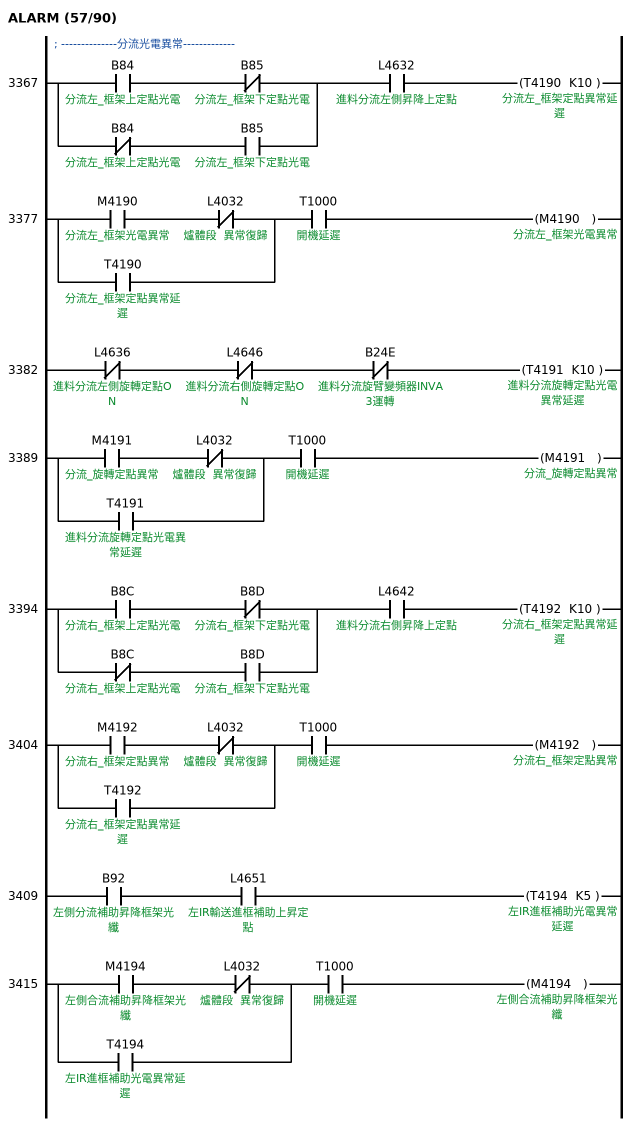
; --------------分流光電異常-------------
3367  LD      B84  ; 分流左_框架上定點光電
      ANI     B85  ; 分流左_框架下定點光電
      LDI     B84  ; 分流左_框架上定點光電
      AND     B85  ; 分流左_框架下定點光電
      ORB
      AND     L4632  ; 進料分流左側昇降上定點
      OUT     T4190 K10  ; 分流左_框架定點異常延遲
3377  LD      M4190  ; 分流左_框架光電異常
      ANI     L4032  ; 爐體段  異常復歸
      OR      T4190  ; 分流左_框架定點異常延遲
      AND     T1000  ; 開機延遲
      OUT     M4190  ; 分流左_框架光電異常
3382  LDI     L4636  ; 進料分流左側旋轉定點ON
      ANI     L4646  ; 進料分流右側旋轉定點ON
      ANI     B24E  ; 進料分流旋臂變頻器INVA3運轉
      OUT     T4191 K10  ; 進料分流旋轉定點光電異常延遲
3389  LD      M4191  ; 分流_旋轉定點異常
      ANI     L4032  ; 爐體段  異常復歸
      OR      T4191  ; 進料分流旋轉定點光電異常延遲
      AND     T1000  ; 開機延遲
      OUT     M4191  ; 分流_旋轉定點異常
3394  LD      B8C  ; 分流右_框架上定點光電
      ANI     B8D  ; 分流右_框架下定點光電
      LDI     B8C  ; 分流右_框架上定點光電
      AND     B8D  ; 分流右_框架下定點光電
      ORB
      AND     L4642  ; 進料分流右側昇降上定點
      OUT     T4192 K10  ; 分流右_框架定點異常延遲
3404  LD      M4192  ; 分流右_框架定點異常
      ANI     L4032  ; 爐體段  異常復歸
      OR      T4192  ; 分流右_框架定點異常延遲
      AND     T1000  ; 開機延遲
      OUT     M4192  ; 分流右_框架定點異常
3409  LD      B92  ; 左側分流補助昇降框架光纖
      AND     L4651  ; 左IR輸送進框補助上昇定點
      OUT     T4194 K5  ; 左IR進框補助光電異常延遲
3415  LD      M4194  ; 左側合流補助昇降框架光纖
      ANI     L4032  ; 爐體段  異常復歸
      OR      T4194  ; 左IR進框補助光電異常延遲
      AND     T1000  ; 開機延遲
      OUT     M4194  ; 左側合流補助昇降框架光纖
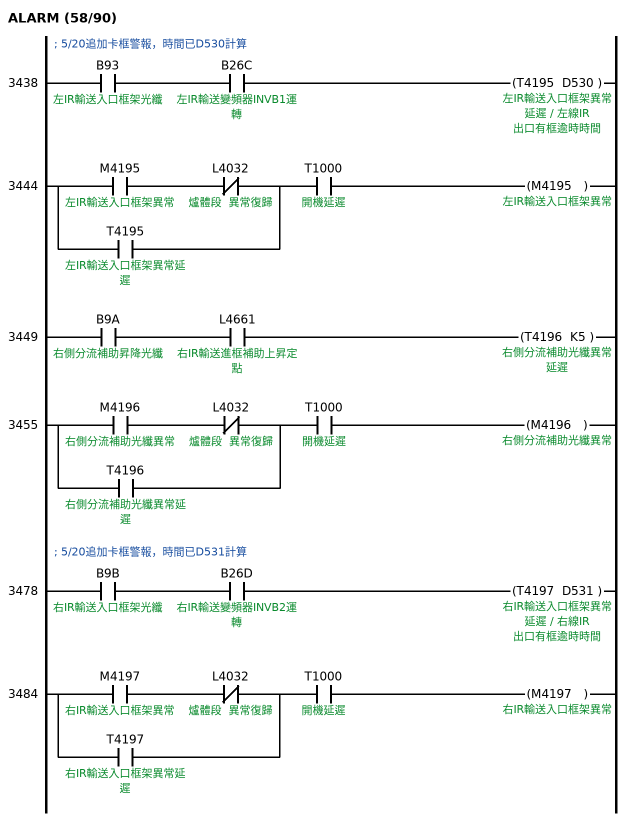
; 5/20追加卡框警報，時間已D530計算
3438  LD      B93  ; 左IR輸送入口框架光纖
      AND     B26C  ; 左IR輸送變頻器INVB1運轉
      OUT     T4195 D530  ; 左IR輸送入口框架異常延遲 / 左線IR  出口有框逾時時間
3444  LD      M4195  ; 左IR輸送入口框架異常
      ANI     L4032  ; 爐體段  異常復歸
      OR      T4195  ; 左IR輸送入口框架異常延遲
      AND     T1000  ; 開機延遲
      OUT     M4195  ; 左IR輸送入口框架異常
3449  LD      B9A  ; 右側分流補助昇降光纖
      AND     L4661  ; 右IR輸送進框補助上昇定點
      OUT     T4196 K5  ; 右側分流補助光纖異常延遲
3455  LD      M4196  ; 右側分流補助光纖異常
      ANI     L4032  ; 爐體段  異常復歸
      OR      T4196  ; 右側分流補助光纖異常延遲
      AND     T1000  ; 開機延遲
      OUT     M4196  ; 右側分流補助光纖異常
; 5/20追加卡框警報，時間已D531計算
3478  LD      B9B  ; 右IR輸送入口框架光纖
      AND     B26D  ; 右IR輸送變頻器INVB2運轉
      OUT     T4197 D531  ; 右IR輸送入口框架異常延遲 / 右線IR  出口有框逾時時間
3484  LD      M4197  ; 右IR輸送入口框架異常
      ANI     L4032  ; 爐體段  異常復歸
      OR      T4197  ; 右IR輸送入口框架異常延遲
      AND     T1000  ; 開機延遲
      OUT     M4197  ; 右IR輸送入口框架異常
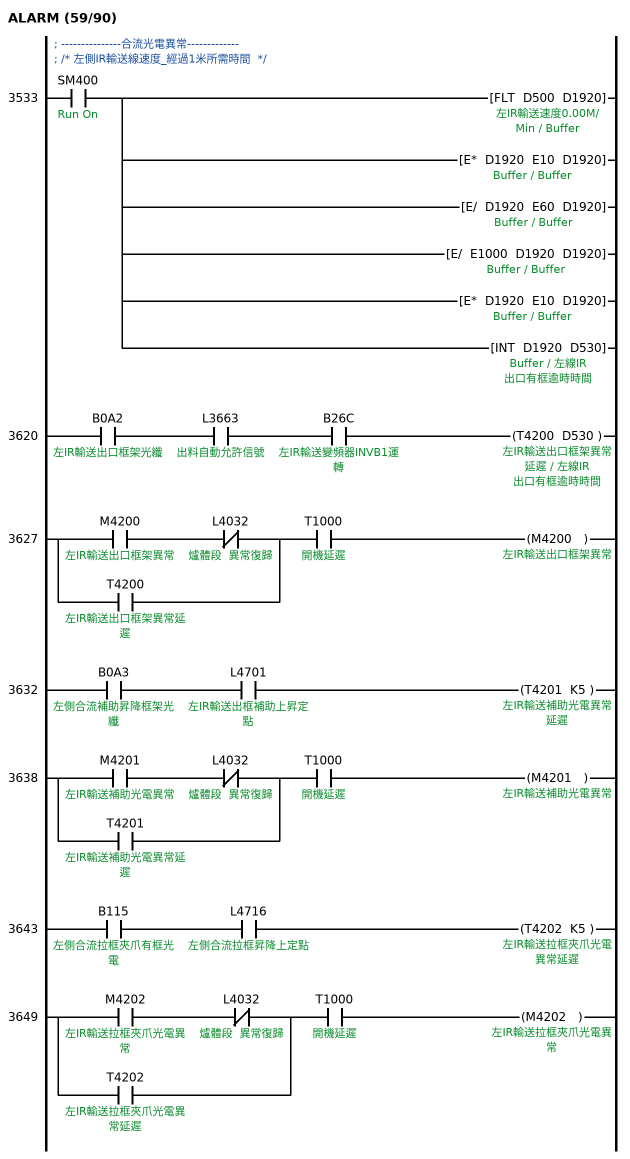
; ---------------合流光電異常-------------
; /* 左側IR輸送線速度_經過1米所需時間  */
3533  LD      SM400  ; Run On
      FLT     D500 D1920  ; 左IR輸送速度0.00M/Min / Buffer
      E*      D1920 E10 D1920
        [note] /* 換算線速度單位_mm/M */
      E/      D1920 E60 D1920
        [note] /* 換算每秒移動距離_單位mm/S */
      E/      E1000 D1920 D1920
        [note] /* 計算每米需移動時間_Sec/M */
      E*      D1920 E10 D1920
        [note] /* 換算時間單位_0.1Sec */
      INT     D1920 D530
3620  LD      B0A2  ; 左IR輸送出口框架光纖
      AND     L3663  ; 出料自動允許信號
      AND     B26C  ; 左IR輸送變頻器INVB1運轉
      OUT     T4200 D530  ; 左IR輸送出口框架異常延遲 / 左線IR  出口有框逾時時間
3627  LD      M4200  ; 左IR輸送出口框架異常
      ANI     L4032  ; 爐體段  異常復歸
      OR      T4200  ; 左IR輸送出口框架異常延遲
      AND     T1000  ; 開機延遲
      OUT     M4200  ; 左IR輸送出口框架異常
3632  LD      B0A3  ; 左側合流補助昇降框架光纖
      AND     L4701  ; 左IR輸送出框補助上昇定點
      OUT     T4201 K5  ; 左IR輸送補助光電異常延遲
3638  LD      M4201  ; 左IR輸送補助光電異常
      ANI     L4032  ; 爐體段  異常復歸
      OR      T4201  ; 左IR輸送補助光電異常延遲
      AND     T1000  ; 開機延遲
      OUT     M4201  ; 左IR輸送補助光電異常
3643  LD      B115  ; 左側合流拉框夾爪有框光電
      AND     L4716  ; 左側合流拉框昇降上定點
      OUT     T4202 K5  ; 左IR輸送拉框夾爪光電異常延遲
3649  LD      M4202  ; 左IR輸送拉框夾爪光電異常
      ANI     L4032  ; 爐體段  異常復歸
      OR      T4202  ; 左IR輸送拉框夾爪光電異常延遲
      AND     T1000  ; 開機延遲
      OUT     M4202  ; 左IR輸送拉框夾爪光電異常
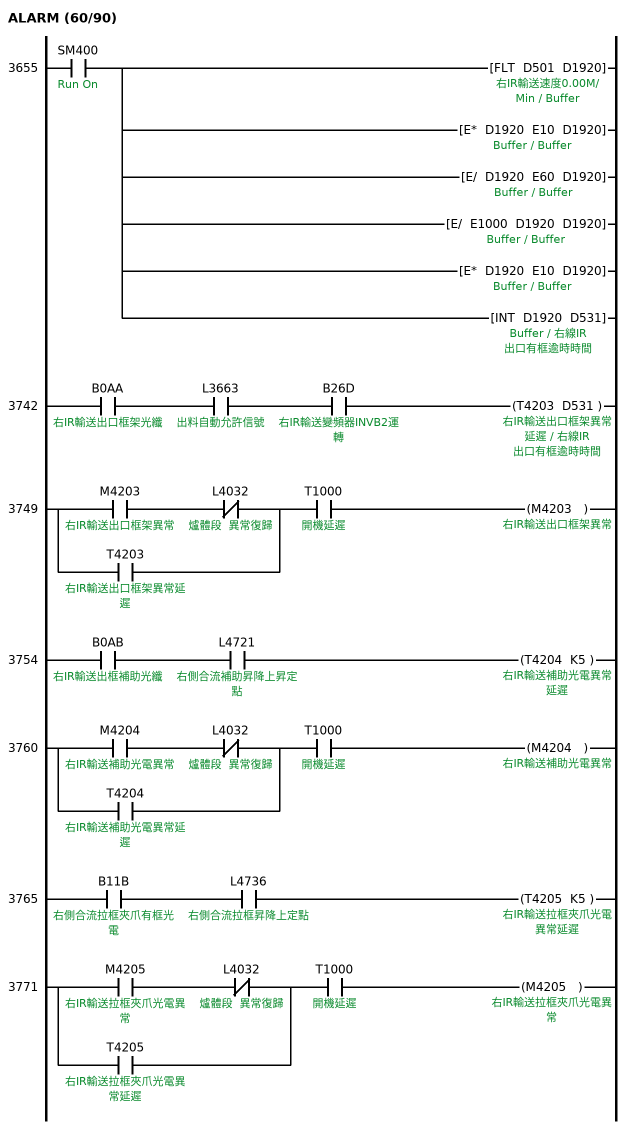
3655  LD      SM400  ; Run On
      FLT     D501 D1920  ; 右IR輸送速度0.00M/Min
      E*      D1920 E10 D1920
        [note] /* 換算線速度單位_mm/M */
      E/      D1920 E60 D1920
        [note] /* 換算每秒移動距離_單位mm/S */
      E/      E1000 D1920 D1920
        [note] /* 計算每米需移動時間_Sec/M */
      E*      D1920 E10 D1920
        [note] /* 換算時間單位_0.1Sec */
      INT     D1920 D531
3742  LD      B0AA  ; 右IR輸送出口框架光纖
      AND     L3663  ; 出料自動允許信號
      AND     B26D  ; 右IR輸送變頻器INVB2運轉
      OUT     T4203 D531  ; 右IR輸送出口框架異常延遲 / 右線IR  出口有框逾時時間
3749  LD      M4203  ; 右IR輸送出口框架異常
      ANI     L4032  ; 爐體段  異常復歸
      OR      T4203  ; 右IR輸送出口框架異常延遲
      AND     T1000  ; 開機延遲
      OUT     M4203  ; 右IR輸送出口框架異常
3754  LD      B0AB  ; 右IR輸送出框補助光纖
      AND     L4721  ; 右側合流補助昇降上昇定點
      OUT     T4204 K5  ; 右IR輸送補助光電異常延遲
3760  LD      M4204  ; 右IR輸送補助光電異常
      ANI     L4032  ; 爐體段  異常復歸
      OR      T4204  ; 右IR輸送補助光電異常延遲
      AND     T1000  ; 開機延遲
      OUT     M4204  ; 右IR輸送補助光電異常
3765  LD      B11B  ; 右側合流拉框夾爪有框光電
      AND     L4736  ; 右側合流拉框昇降上定點
      OUT     T4205 K5  ; 右IR輸送拉框夾爪光電異常延遲
3771  LD      M4205  ; 右IR輸送拉框夾爪光電異常
      ANI     L4032  ; 爐體段  異常復歸
      OR      T4205  ; 右IR輸送拉框夾爪光電異常延遲
      AND     T1000  ; 開機延遲
      OUT     M4205  ; 右IR輸送拉框夾爪光電異常
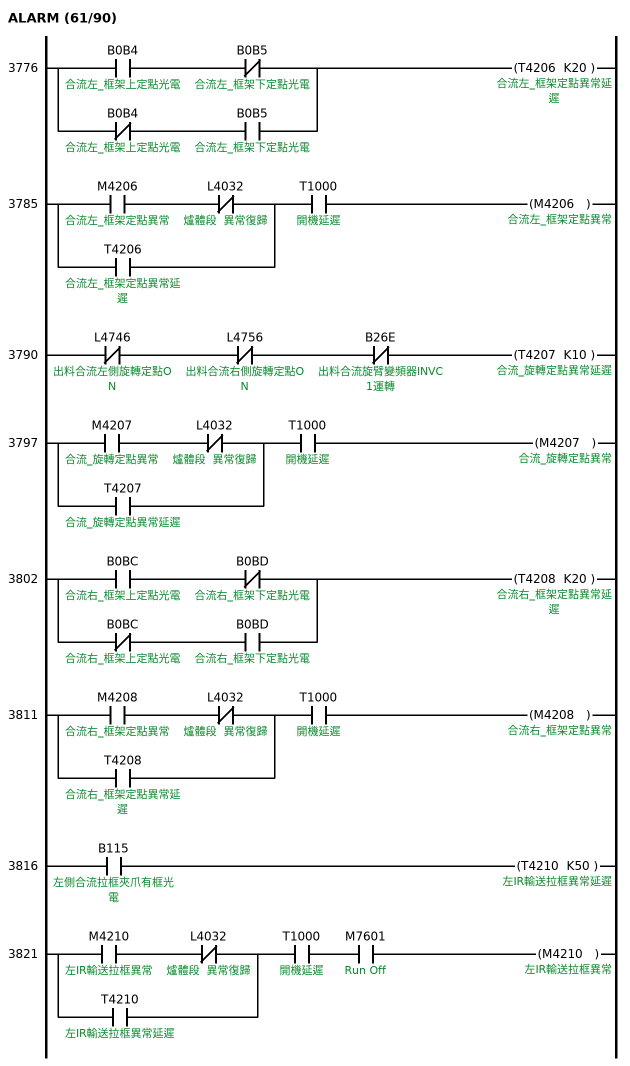
3776  LD      B0B4  ; 合流左_框架上定點光電
      ANI     B0B5  ; 合流左_框架下定點光電
      LDI     B0B4  ; 合流左_框架上定點光電
      AND     B0B5  ; 合流左_框架下定點光電
      ORB
      OUT     T4206 K20  ; 合流左_框架定點異常延遲
3785  LD      M4206  ; 合流左_框架定點異常
      ANI     L4032  ; 爐體段  異常復歸
      OR      T4206  ; 合流左_框架定點異常延遲
      AND     T1000  ; 開機延遲
      OUT     M4206  ; 合流左_框架定點異常
3790  LDI     L4746  ; 出料合流左側旋轉定點ON
      ANI     L4756  ; 出料合流右側旋轉定點ON
      ANI     B26E  ; 出料合流旋臂變頻器INVC1運轉
      OUT     T4207 K10  ; 合流_旋轉定點異常延遲
3797  LD      M4207  ; 合流_旋轉定點異常
      ANI     L4032  ; 爐體段  異常復歸
      OR      T4207  ; 合流_旋轉定點異常延遲
      AND     T1000  ; 開機延遲
      OUT     M4207  ; 合流_旋轉定點異常
3802  LD      B0BC  ; 合流右_框架上定點光電
      ANI     B0BD  ; 合流右_框架下定點光電
      LDI     B0BC  ; 合流右_框架上定點光電
      AND     B0BD  ; 合流右_框架下定點光電
      ORB
      OUT     T4208 K20  ; 合流右_框架定點異常延遲
3811  LD      M4208  ; 合流右_框架定點異常
      ANI     L4032  ; 爐體段  異常復歸
      OR      T4208  ; 合流右_框架定點異常延遲
      AND     T1000  ; 開機延遲
      OUT     M4208  ; 合流右_框架定點異常
3816  LD      B115  ; 左側合流拉框夾爪有框光電
      OUT     T4210 K50  ; 左IR輸送拉框異常延遲
3821  LD      M4210  ; 左IR輸送拉框異常
      ANI     L4032  ; 爐體段  異常復歸
      OR      T4210  ; 左IR輸送拉框異常延遲
      AND     T1000  ; 開機延遲
      AND     M7601  ; Run Off
      OUT     M4210  ; 左IR輸送拉框異常
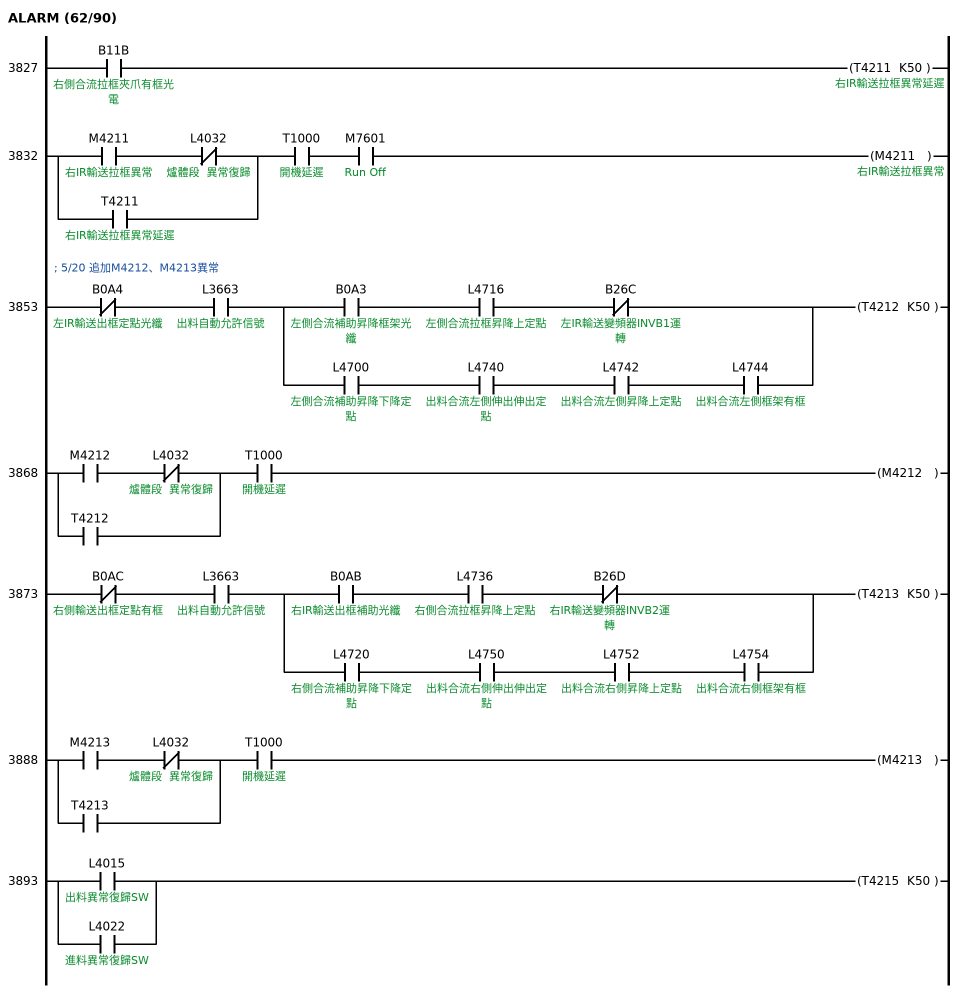
3827  LD      B11B  ; 右側合流拉框夾爪有框光電
      OUT     T4211 K50  ; 右IR輸送拉框異常延遲
3832  LD      M4211  ; 右IR輸送拉框異常
      ANI     L4032  ; 爐體段  異常復歸
      OR      T4211  ; 右IR輸送拉框異常延遲
      AND     T1000  ; 開機延遲
      AND     M7601  ; Run Off
      OUT     M4211  ; 右IR輸送拉框異常
; 5/20 追加M4212、M4213異常
3853  LDI     B0A4  ; 左IR輸送出框定點光纖
      AND     L3663  ; 出料自動允許信號
      LD      B0A3  ; 左側合流補助昇降框架光纖
      AND     L4716  ; 左側合流拉框昇降上定點
      ANI     B26C  ; 左IR輸送變頻器INVB1運轉
      LD      L4700  ; 左側合流補助昇降下降定點
      AND     L4740  ; 出料合流左側伸出伸出定點
      AND     L4742  ; 出料合流左側昇降上定點
      AND     L4744  ; 出料合流左側框架有框
      ORB
      ANB
      OUT     T4212 K50
3868  LD      M4212
      ANI     L4032  ; 爐體段  異常復歸
      OR      T4212
      AND     T1000  ; 開機延遲
      OUT     M4212
3873  LDI     B0AC  ; 右側輸送出框定點有框
      AND     L3663  ; 出料自動允許信號
      LD      B0AB  ; 右IR輸送出框補助光纖
      AND     L4736  ; 右側合流拉框昇降上定點
      ANI     B26D  ; 右IR輸送變頻器INVB2運轉
      LD      L4720  ; 右側合流補助昇降下降定點
      AND     L4750  ; 出料合流右側伸出伸出定點
      AND     L4752  ; 出料合流右側昇降上定點
      AND     L4754  ; 出料合流右側框架有框
      ORB
      ANB
      OUT     T4213 K50
3888  LD      M4213
      ANI     L4032  ; 爐體段  異常復歸
      OR      T4213
      AND     T1000  ; 開機延遲
      OUT     M4213
3893  LD      L4015  ; 出料異常復歸SW
      OR      L4022  ; 進料異常復歸SW
      OUT     T4215 K50
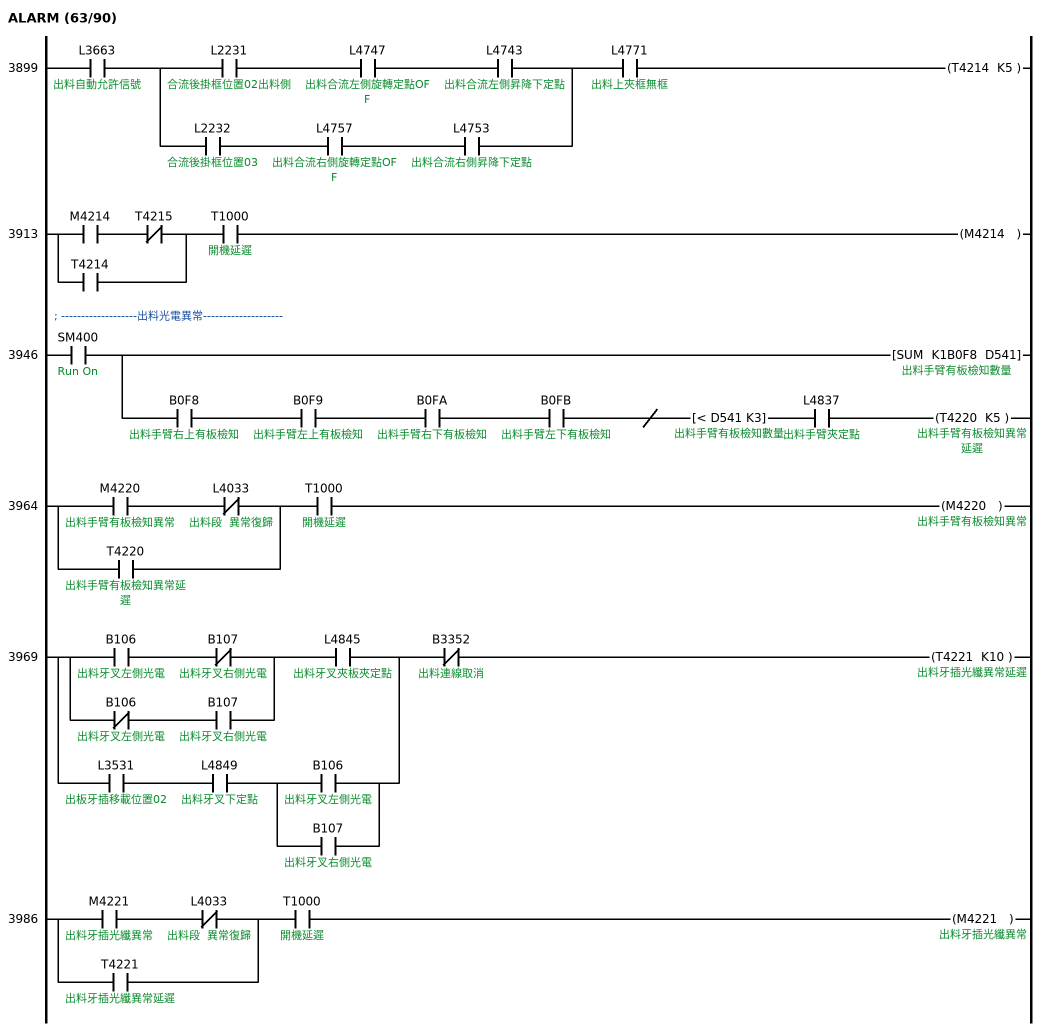
3899  LD      L3663  ; 出料自動允許信號
      LD      L2231  ; 合流後掛框位置02出料側
      AND     L4747  ; 出料合流左側旋轉定點OFF
      AND     L4743  ; 出料合流左側昇降下定點
      LD      L2232  ; 合流後掛框位置03
      AND     L4757  ; 出料合流右側旋轉定點OFF
      AND     L4753  ; 出料合流右側昇降下定點
      ORB
      ANB
      AND     L4771  ; 出料上夾框無框
      OUT     T4214 K5
3913  LD      M4214
      ANI     T4215
      OR      T4214
      AND     T1000  ; 開機延遲
      OUT     M4214
; -------------------出料光電異常--------------------
3946  LD      SM400  ; Run On
      SUM     K1B0F8 D541  ; 出料手臂右上有板檢知 / 出料手臂有板檢知數量
      AND     B0F8  ; 出料手臂右上有板檢知
      AND     B0F9  ; 出料手臂左上有板檢知
      AND     B0FA  ; 出料手臂右下有板檢知
      AND     B0FB  ; 出料手臂左下有板檢知
      INV
      AND<    D541 K3  ; 出料手臂有板檢知數量
      AND     L4837  ; 出料手臂夾定點
      OUT     T4220 K5  ; 出料手臂有板檢知異常延遲
3964  LD      M4220  ; 出料手臂有板檢知異常
      ANI     L4033  ; 出料段  異常復歸
      OR      T4220  ; 出料手臂有板檢知異常延遲
      AND     T1000  ; 開機延遲
      OUT     M4220  ; 出料手臂有板檢知異常
3969  LD      B106  ; 出料牙叉左側光電
      ANI     B107  ; 出料牙叉右側光電
      LDI     B106  ; 出料牙叉左側光電
      AND     B107  ; 出料牙叉右側光電
      ORB
      AND     L4845  ; 出料牙叉夾板夾定點
      LD      L3531  ; 出板牙插移載位置02
      AND     L4849  ; 出料牙叉下定點
      LD      B106  ; 出料牙叉左側光電
      OR      B107  ; 出料牙叉右側光電
      ANB
      ORB
      ANI     B3352  ; 出料連線取消
      OUT     T4221 K10  ; 出料牙插光纖異常延遲
3986  LD      M4221  ; 出料牙插光纖異常
      ANI     L4033  ; 出料段  異常復歸
      OR      T4221  ; 出料牙插光纖異常延遲
      AND     T1000  ; 開機延遲
      OUT     M4221  ; 出料牙插光纖異常
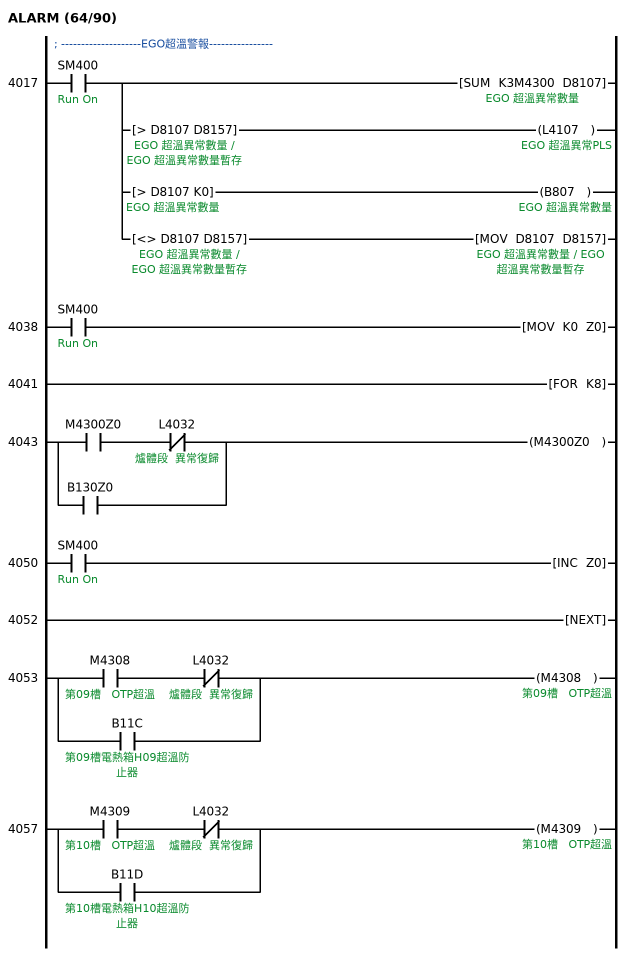
; --------------------EGO超溫警報----------------
4017  LD      SM400  ; Run On
      SUM     K3M4300 D8107  ; 第01槽   OTP超溫 / EGO 超溫異常數量
      MPS
      AND>    D8107 D8157  ; EGO 超溫異常數量 / EGO 超溫異常數量暫存
      OUT     L4107  ; EGO 超溫異常PLS
      MRD
      AND>    D8107 K0  ; EGO 超溫異常數量
      OUT     B807  ; EGO 超溫異常數量
      MPP
      AND<>   D8107 D8157  ; EGO 超溫異常數量 / EGO 超溫異常數量暫存
      MOV     D8107 D8157
4038  LD      SM400  ; Run On
      MOV     K0 Z0
4041  FOR     K8
4043  LD      M4300Z0
      ANI     L4032  ; 爐體段  異常復歸
      OR      B130Z0
      OUT     M4300Z0
4050  LD      SM400  ; Run On
      INC     Z0
4052  NEXT
4053  LD      M4308  ; 第09槽   OTP超溫
      ANI     L4032  ; 爐體段  異常復歸
      OR      B11C  ; 第09槽電熱箱H09超溫防止器
      OUT     M4308  ; 第09槽   OTP超溫
4057  LD      M4309  ; 第10槽   OTP超溫
      ANI     L4032  ; 爐體段  異常復歸
      OR      B11D  ; 第10槽電熱箱H10超溫防止器
      OUT     M4309  ; 第10槽   OTP超溫
